KUKA KRL program: EPS_2_251580_SMH02_A_20251111081754.src

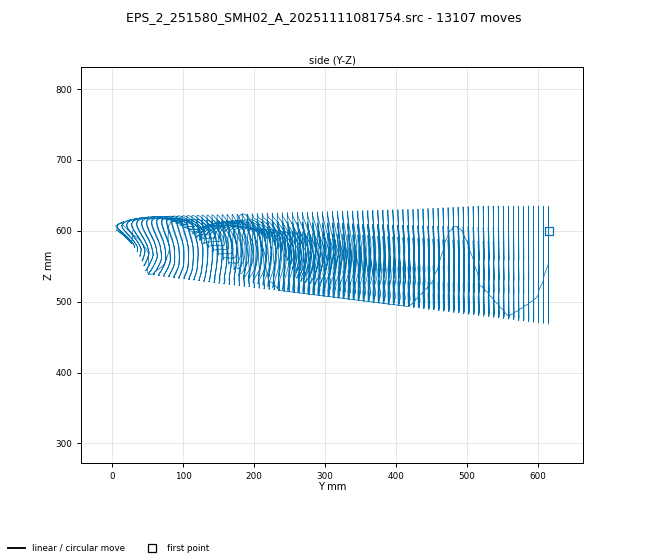
[picture p0: tool path of EPS_2_251580_SMH02_A_20251111081754.src, 13107 of 13109 moves have a stored position in this frame; points joined in program order, loops and branches not executed]
&ACCESS RVP
&REL 4
&COMMENT QRS 19112012
&PARAM EDITMASK = *
DEF PART()
EXT BAS (BAS_COMMAND :IN,REAL :IN )
INT I
BAS (#INITMOV,0 )

;KUKA QRS Post kuka4.cps  Date:22-06-2017 !

File_ID=2902

QRS_PRE_INIT()

;Init var - Until changes are made in qrs_pre_init
Outlet_Square_prg=0
Inlet_1_Square_prg=0
Inlet_2_Square_prg=0
Inlet_3_Square_prg=0
Inlet_4_Square_prg=0
Inlet_5_Square_prg=0

Outlet_1={X 0.000, Y 520.000, Z 560.000, B 0.000, E1 0.000 }
Inlet_1={X 0.000, Y 523.590, Z 510.000, B 0.000, E1 90.000 }
Inlet_2={X 0.000, Y 522.160, Z 530.000, B 0.000, E1 146.000 }
Outlet_1_type=150
Inlet_1_type=150
Inlet_2_type=150
;QRS#1=Sidecore dimensions
;QRS#2=150-6" PVC SDR 28
;QRS#3=150-6" PVC SDR 28
;QRS#4=150-6" PVC SDR 28
;QRS#5=
;QRS#6=
;QRS#7=
;QRS#8=
;QRS#9=10-06 PSX
;QRS#10=10-06 PSX
;QRS#11=10-06 PSX
;QRS#12=
;QRS#13=
;QRS#14=
;QRS#15=
;QRS#16=1220x127x914 3'
;QRS#17=EPS Height
;QRS#18=635
;QRS#19=*
;QRS#20= UPDATED VERSION 22-06-2017
;QRS#21=*
Outlet_Square=070
Inlet_1_Square=070
Inlet_2_Square=070
Inlet_3_Square=0
Inlet_4_Square=0
Inlet_5_Square=0
Mill_Square=1
Outlet_Square_Prg=203
Inlet_1_Square_prg=203
Inlet_2_Square_prg=203

QRS_INIT()

$ADVANCE=5

; T1
PTP {E1 173.473,E2 173.473}
PTP {X 0,Y 615.499,A -85,B 0,C 180,E1 173.473,E2 173.473,E3 0,E4 0,E5 0,E6 0}
QRS_SPEED_INIT()
LIN {X 0,Y 615.499,Z 600,A -85,B 0,C 180,E1 173.473,E2 173.473,E3 0,E4 0,E5 0,E6 0} C_VEL
LIN {X 0,Y 615.499,Z 569.968,A -85,B 0,C 180,E1 173.473,E2 173.473} C_VEL
LIN {X 0,Y 615.499,Z 557.271,A -85,B 0,C 180,E1 173.473,E2 173.473} C_VEL
LIN {X 0,Y 615.498,Z 555.824,A -85,B 0,C 180,E1 173.416,E2 173.416} C_VEL
LIN {X 0,Y 615.496,Z 547.552,A -85,B 0,C 180,E1 172.702,E2 172.702} C_VEL
LIN {X 0,Y 615.476,Z 537.678,A -85,B 0,C 180,E1 172.042,E2 172.042} C_VEL
LIN {X 0,Y 615.489,Z 529.919,A -85,B 0,C 180,E1 171.629,E2 171.629} C_VEL
LIN {X 0,Y 615.493,Z 521.057,A -85,B 0,C 180,E1 171.257,E2 171.257} C_VEL
LIN {X 0,Y 615.492,Z 511.835,A -85,B 0,C 180,E1 170.967,E2 170.967} C_VEL
LIN {X 0,Y 615.489,Z 506.039,A -85,B 0,C 180,E1 170.822,E2 170.822} C_VEL
LIN {X 0,Y 615.478,Z 501.144,A -85,B 0,C 180,E1 168.139,E2 168.139} C_VEL
LIN {X 0,Y 615.493,Z 496.29,A -85,B 0,C 180,E1 165.451,E2 165.451} C_VEL
LIN {X 0,Y 615.49,Z 491.434,A -85,B 0,C 180,E1 162.73,E2 162.73} C_VEL
LIN {X 0,Y 615.491,Z 486.577,A -85,B 0,C 180,E1 159.967,E2 159.967} C_VEL
LIN {X 0,Y 615.477,Z 481.72,A -85,B 0,C 180,E1 157.155,E2 157.155} C_VEL
LIN {X 0,Y 615.486,Z 477.105,A -85,B 0,C 180,E1 154.432,E2 154.432} C_VEL
LIN {X 0,Y 615.496,Z 474.066,A -85,B 0,C 180,E1 152.501,E2 152.501} C_VEL
LIN {X 0,Y 615.489,Z 480.62,A -85,B 0,C 180,E1 149.84,E2 149.84} C_VEL
LIN {X 0,Y 615.489,Z 486.401,A -85,B 0,C 180,E1 147.543,E2 147.543} C_VEL
LIN {X 0,Y 615.488,Z 493.466,A -85,B 0,C 180,E1 144.785,E2 144.785} C_VEL
LIN {X 0,Y 615.484,Z 500.912,A -85,B 0,C 180,E1 141.931,E2 141.931} C_VEL
LIN {X 0,Y 615.483,Z 507.646,A -85,B 0,C 180,E1 139.393,E2 139.393} C_VEL
LIN {X 0,Y 615.497,Z 514.698,A -85,B 0,C 180,E1 136.756,E2 136.756} C_VEL
LIN {X 0,Y 615.483,Z 522.177,A -85,B 0,C 180,E1 133.997,E2 133.997} C_VEL
LIN {X 0,Y 615.485,Z 524.739,A -85,B 0,C 180,E1 133.109,E2 133.109} C_VEL
LIN {X 0,Y 615.497,Z 537.239,A -85,B 0,C 180,E1 132.785,E2 132.785} C_VEL
LIN {X 0,Y 615.477,Z 546.369,A -85,B 0,C 180,E1 132.441,E2 132.441} C_VEL
LIN {X 0,Y 615.481,Z 555.26,A -85,B 0,C 180,E1 132.003,E2 132.003} C_VEL
LIN {X 0,Y 615.489,Z 562.693,A -85,B 0,C 180,E1 131.549,E2 131.549} C_VEL
LIN {X 0,Y 615.499,Z 570.437,A -85,B 0,C 180,E1 130.972,E2 130.972} C_VEL
LIN {X 0,Y 615.495,Z 577.327,A -85,B 0,C 180,E1 130.348,E2 130.348} C_VEL
LIN {X 0,Y 615.498,Z 584.294,A -85,B 0,C 180,E1 129.577,E2 129.577} C_VEL
LIN {X 0,Y 615.497,Z 590.588,A -85,B 0,C 180,E1 128.694,E2 128.694} C_VEL
LIN {X 0,Y 615.495,Z 594.491,A -85,B 0,C 180,E1 128.013,E2 128.013} C_VEL
LIN {X 0,Y 615.492,Z 598.012,A -85,B 0,C 180,E1 127.242,E2 127.242} C_VEL
LIN {X 0,Y 615.49,Z 600.84,A -85,B 0,C 180,E1 126.425,E2 126.425} C_VEL
LIN {X 0,Y 615.493,Z 602.8,A -85,B 0,C 180,E1 125.616,E2 125.616} C_VEL
LIN {X 0,Y 615.498,Z 604.058,A -85,B 0,C 180,E1 124.702,E2 124.702} C_VEL
LIN {X 0,Y 615.493,Z 604.378,A -85,B 0,C 180,E1 124.022,E2 124.022} C_VEL
LIN {X 0,Y 615.494,Z 604.074,A -85,B 0,C 180,E1 123.236,E2 123.236} C_VEL
LIN {X 0,Y 615.489,Z 602.87,A -85,B 0,C 180,E1 122.331,E2 122.331} C_VEL
LIN {X 0,Y 615.495,Z 601.344,A -85,B 0,C 180,E1 121.685,E2 121.685} C_VEL
LIN {X 0,Y 615.489,Z 597.454,A -85,B 0,C 180,E1 120.539,E2 120.539} C_VEL
LIN {X 0,Y 615.494,Z 592.819,A -85,B 0,C 180,E1 119.601,E2 119.601} C_VEL
LIN {X 0,Y 615.499,Z 588.063,A -85,B 0,C 180,E1 118.844,E2 118.844} C_VEL
LIN {X 0,Y 615.497,Z 583.01,A -85,B 0,C 180,E1 118.183,E2 118.183} C_VEL
LIN {X 0,Y 615.497,Z 577.153,A -85,B 0,C 180,E1 117.545,E2 117.545} C_VEL
LIN {X 0,Y 615.498,Z 569.916,A -85,B 0,C 180,E1 116.895,E2 116.895} C_VEL
LIN {X 0,Y 615.478,Z 562.594,A -85,B 0,C 180,E1 116.354,E2 116.354} C_VEL
LIN {X 0,Y 615.488,Z 553.468,A -85,B 0,C 180,E1 115.807,E2 115.807} C_VEL
LIN {X 0,Y 615.485,Z 541.734,A -85,B 0,C 180,E1 115.28,E2 115.28} C_VEL
LIN {X 0,Y 615.496,Z 532.824,A -85,B 0,C 180,E1 114.992,E2 114.992} C_VEL
LIN {X 0,Y 615.494,Z 524.808,A -85,B 0,C 180,E1 114.789,E2 114.789} C_VEL
LIN {X 0,Y 615.482,Z 518.038,A -85,B 0,C 180,E1 112.137,E2 112.137} C_VEL
LIN {X 0,Y 615.485,Z 510.962,A -85,B 0,C 180,E1 109.338,E2 109.338} C_VEL
LIN {X 0,Y 615.48,Z 504.089,A -85,B 0,C 180,E1 106.587,E2 106.587} C_VEL
LIN {X 0,Y 615.495,Z 497.407,A -85,B 0,C 180,E1 103.874,E2 103.874} C_VEL
LIN {X 0,Y 615.486,Z 490.182,A -85,B 0,C 180,E1 100.887,E2 100.887} C_VEL
LIN {X 0,Y 615.483,Z 484.608,A -85,B 0,C 180,E1 98.537,E2 98.537} C_VEL
LIN {X 0,Y 615.493,Z 478.479,A -85,B 0,C 180,E1 95.899,E2 95.899} C_VEL
LIN {X 0,Y 615.481,Z 472.517,A -85,B 0,C 180,E1 93.273,E2 93.273} C_VEL
LIN {X 0,Y 615.478,Z 468.511,A -85,B 0,C 180,E1 91.473,E2 91.473} C_VEL
LIN {X 0,Y 615.48,Z 468.51,A -85,B 0,C 180,E1 88.692,E2 88.692} C_VEL
LIN {X 0,Y 615.488,Z 468.512,A -85,B 0,C 180,E1 86.072,E2 86.072} C_VEL
LIN {X 0,Y 615.49,Z 468.512,A -85,B 0,C 180,E1 83.42,E2 83.42} C_VEL
LIN {X 0,Y 615.48,Z 468.511,A -85,B 0,C 180,E1 80.801,E2 80.801} C_VEL
LIN {X 0,Y 615.49,Z 468.508,A -85,B 0,C 180,E1 78.14,E2 78.14} C_VEL
LIN {X 0,Y 615.487,Z 468.512,A -85,B 0,C 180,E1 75.451,E2 75.451} C_VEL
LIN {X 0,Y 615.488,Z 468.511,A -85,B 0,C 180,E1 72.73,E2 72.73} C_VEL
LIN {X 0,Y 615.488,Z 468.508,A -85,B 0,C 180,E1 69.968,E2 69.968} C_VEL
LIN {X 0,Y 615.489,Z 468.512,A -85,B 0,C 180,E1 67.156,E2 67.156} C_VEL
LIN {X 0,Y 615.495,Z 468.507,A -85,B 0,C 180,E1 64.285,E2 64.285} C_VEL
LIN {X 0,Y 615.484,Z 468.511,A -85,B 0,C 180,E1 61.342,E2 61.342} C_VEL
LIN {X 0,Y 615.495,Z 468.51,A -85,B 0,C 180,E1 58.913,E2 58.913} C_VEL
LIN {X 0,Y 615.49,Z 468.513,A -85,B 0,C 180,E1 56.466,E2 56.466} C_VEL
LIN {X 0,Y 615.494,Z 468.511,A -85,B 0,C 180,E1 54.166,E2 54.166} C_VEL
LIN {X 0,Y 615.493,Z 468.509,A -85,B 0,C 180,E1 51.932,E2 51.932} C_VEL
LIN {X 0,Y 615.485,Z 468.514,A -85,B 0,C 180,E1 49.394,E2 49.394} C_VEL
LIN {X 0,Y 615.492,Z 468.511,A -85,B 0,C 180,E1 46.756,E2 46.756} C_VEL
LIN {X 0,Y 615.484,Z 468.509,A -85,B 0,C 180,E1 43.998,E2 43.998} C_VEL
LIN {X 0,Y 615.495,Z 468.512,A -85,B 0,C 180,E1 41.096,E2 41.096} C_VEL
LIN {X 0,Y 615.481,Z 468.512,A -85,B 0,C 180,E1 38.905,E2 38.905} C_VEL
LIN {X 0,Y 615.488,Z 468.512,A -85,B 0,C 180,E1 36.425,E2 36.425} C_VEL
LIN {X 0,Y 615.485,Z 468.509,A -85,B 0,C 180,E1 33.535,E2 33.535} C_VEL
LIN {X 0,Y 615.479,Z 468.51,A -85,B 0,C 180,E1 30.92,E2 30.92} C_VEL
LIN {X 0,Y 615.492,Z 468.507,A -85,B 0,C 180,E1 28.452,E2 28.452} C_VEL
LIN {X 0,Y 615.495,Z 468.512,A -85,B 0,C 180,E1 25.571,E2 25.571} C_VEL
LIN {X 0,Y 615.48,Z 468.51,A -85,B 0,C 180,E1 22.845,E2 22.845} C_VEL
LIN {X 0,Y 615.488,Z 468.51,A -85,B 0,C 180,E1 20.033,E2 20.033} C_VEL
LIN {X 0,Y 615.49,Z 468.512,A -85,B 0,C 180,E1 17.27,E2 17.27} C_VEL
LIN {X 0,Y 615.494,Z 468.507,A -85,B 0,C 180,E1 14.549,E2 14.549} C_VEL
LIN {X 0,Y 615.48,Z 468.511,A -85,B 0,C 180,E1 11.861,E2 11.861} C_VEL
LIN {X 0,Y 615.486,Z 468.514,A -85,B 0,C 180,E1 9.199,E2 9.199} C_VEL
LIN {X 0,Y 615.497,Z 468.509,A -85,B 0,C 180,E1 6.557,E2 6.557} C_VEL
LIN {X 0,Y 615.479,Z 468.51,A -85,B 0,C 180,E1 3.929,E2 3.929} C_VEL
LIN {X 0,Y 615.487,Z 468.508,A -85,B 0,C 180,E1 1.309,E2 1.309} C_VEL
LIN {X 0,Y 615.485,Z 468.512,A -85,B 0,C 180,E1 -1.309,E2 -1.309} C_VEL
LIN {X 0,Y 615.489,Z 468.514,A -85,B 0,C 180,E1 -3.928,E2 -3.928} C_VEL
LIN {X 0,Y 615.491,Z 468.508,A -85,B 0,C 180,E1 -6.584,E2 -6.584} C_VEL
LIN {X 0,Y 615.483,Z 468.509,A -85,B 0,C 180,E1 -9.199,E2 -9.199} C_VEL
LIN {X 0,Y 615.488,Z 468.51,A -85,B 0,C 180,E1 -11.861,E2 -11.861} C_VEL
LIN {X 0,Y 615.491,Z 468.514,A -85,B 0,C 180,E1 -14.549,E2 -14.549} C_VEL
LIN {X 0,Y 615.495,Z 468.507,A -85,B 0,C 180,E1 -17.27,E2 -17.27} C_VEL
LIN {X 0,Y 615.479,Z 468.511,A -85,B 0,C 180,E1 -20.033,E2 -20.033} C_VEL
LIN {X 0,Y 615.493,Z 468.512,A -85,B 0,C 180,E1 -22.844,E2 -22.844} C_VEL
LIN {X 0,Y 615.48,Z 468.51,A -85,B 0,C 180,E1 -25.716,E2 -25.716} C_VEL
LIN {X 0,Y 615.492,Z 468.514,A -85,B 0,C 180,E1 -28.658,E2 -28.658} C_VEL
LIN {X 0,Y 615.49,Z 468.514,A -85,B 0,C 180,E1 -31.087,E2 -31.087} C_VEL
LIN {X 0,Y 615.486,Z 468.513,A -85,B 0,C 180,E1 -33.535,E2 -33.535} C_VEL
LIN {X 0,Y 615.488,Z 468.508,A -85,B 0,C 180,E1 -36.425,E2 -36.425} C_VEL
LIN {X 0,Y 615.482,Z 468.512,A -85,B 0,C 180,E1 -39.062,E2 -39.062} C_VEL
LIN {X 0,Y 615.494,Z 468.51,A -85,B 0,C 180,E1 -41.473,E2 -41.473} C_VEL
LIN {X 0,Y 615.492,Z 468.512,A -85,B 0,C 180,E1 -44.149,E2 -44.149} C_VEL
LIN {X 0,Y 615.485,Z 468.509,A -85,B 0,C 180,E1 -46.953,E2 -46.953} C_VEL
LIN {X 0,Y 615.498,Z 468.512,A -85,B 0,C 180,E1 -49.91,E2 -49.91} C_VEL
LIN {X 0,Y 615.481,Z 468.51,A -85,B 0,C 180,E1 -52.758,E2 -52.758} C_VEL
LIN {X 0,Y 615.495,Z 468.506,A -85,B 0,C 180,E1 -55.298,E2 -55.298} C_VEL
LIN {X 0,Y 615.477,Z 468.51,A -85,B 0,C 180,E1 -57.671,E2 -57.671} C_VEL
LIN {X 0,Y 615.492,Z 468.707,A -85,B 0,C 180,E1 -59.081,E2 -59.081} C_VEL
LIN {X 0,Y 615.477,Z 477.608,A -85,B 0,C 180,E1 -61.552,E2 -61.552} C_VEL
LIN {X 0,Y 615.489,Z 487.691,A -85,B 0,C 180,E1 -64.285,E2 -64.285} C_VEL
LIN {X 0,Y 615.489,Z 498.525,A -85,B 0,C 180,E1 -67.156,E2 -67.156} C_VEL
LIN {X 0,Y 615.485,Z 509.354,A -85,B 0,C 180,E1 -69.968,E2 -69.968} C_VEL
LIN {X 0,Y 615.477,Z 520.179,A -85,B 0,C 180,E1 -72.73,E2 -72.73} C_VEL
LIN {X 0,Y 615.493,Z 530.988,A -85,B 0,C 180,E1 -75.451,E2 -75.451} C_VEL
LIN {X 0,Y 615.488,Z 541.8,A -85,B 0,C 180,E1 -78.14,E2 -78.14} C_VEL
LIN {X 0,Y 615.481,Z 552.598,A -85,B 0,C 180,E1 -80.801,E2 -80.801} C_VEL
LIN {X 0,Y 615.495,Z 566.17,A -85,B 0,C 180,E1 -81.133,E2 -81.133} C_VEL
LIN {X 0,Y 615.479,Z 575.233,A -85,B 0,C 180,E1 -81.464,E2 -81.464} C_VEL
LIN {X 0,Y 615.487,Z 583.917,A -85,B 0,C 180,E1 -81.877,E2 -81.877} C_VEL
LIN {X 0,Y 615.48,Z 592.206,A -85,B 0,C 180,E1 -82.372,E2 -82.372} C_VEL
LIN {X 0,Y 615.499,Z 599.937,A -85,B 0,C 180,E1 -82.942,E2 -82.942} C_VEL
LIN {X 0,Y 615.498,Z 605.649,A -85,B 0,C 180,E1 -83.444,E2 -83.444} C_VEL
LIN {X 0,Y 615.499,Z 611.924,A -85,B 0,C 180,E1 -84.102,E2 -84.102} C_VEL
LIN {X 0,Y 615.496,Z 617.138,A -85,B 0,C 180,E1 -84.759,E2 -84.759} C_VEL
LIN {X 0,Y 615.497,Z 621.484,A -85,B 0,C 180,E1 -85.416,E2 -85.416} C_VEL
LIN {X 0,Y 615.492,Z 626.605,A -85,B 0,C 180,E1 -86.4,E2 -86.4} C_VEL
LIN {X 0,Y 615.494,Z 629.221,A -85,B 0,C 180,E1 -87.055,E2 -87.055} C_VEL
LIN {X 0,Y 615.497,Z 632.086,A -85,B 0,C 180,E1 -88.037,E2 -88.037} C_VEL
LIN {X 0,Y 615.494,Z 633.33,A -85,B 0,C 180,E1 -88.692,E2 -88.692} C_VEL
LIN {X 0,Y 615.494,Z 634.104,A -85,B 0,C 180,E1 -89.346,E2 -89.346} C_VEL
LIN {X 0,Y 615.491,Z 634.389,A -85,B 0,C 180,E1 -90,E2 -90} C_VEL
LIN {X 0,Y 615.494,Z 634.104,A -85,B 0,C 180,E1 -90.655,E2 -90.655} C_VEL
LIN {X 0,Y 615.494,Z 633.329,A -85,B 0,C 180,E1 -91.309,E2 -91.309} C_VEL
LIN {X 0,Y 615.497,Z 632.085,A -85,B 0,C 180,E1 -91.963,E2 -91.963} C_VEL
LIN {X 0,Y 615.494,Z 629.218,A -85,B 0,C 180,E1 -92.946,E2 -92.946} C_VEL
LIN {X 0,Y 615.492,Z 626.602,A -85,B 0,C 180,E1 -93.601,E2 -93.601} C_VEL
LIN {X 0,Y 615.496,Z 621.48,A -85,B 0,C 180,E1 -94.585,E2 -94.585} C_VEL
LIN {X 0,Y 615.495,Z 615.966,A -85,B 0,C 180,E1 -95.406,E2 -95.406} C_VEL
LIN {X 0,Y 615.498,Z 609.015,A -85,B 0,C 180,E1 -96.228,E2 -96.228} C_VEL
LIN {X 0,Y 615.498,Z 601.856,A -85,B 0,C 180,E1 -96.901,E2 -96.901} C_VEL
LIN {X 0,Y 615.477,Z 594.619,A -85,B 0,C 180,E1 -97.463,E2 -97.463} C_VEL
LIN {X 0,Y 615.492,Z 586.863,A -85,B 0,C 180,E1 -97.958,E2 -97.958} C_VEL
LIN {X 0,Y 615.478,Z 578.911,A -85,B 0,C 180,E1 -98.372,E2 -98.372} C_VEL
LIN {X 0,Y 615.485,Z 569.748,A -85,B 0,C 180,E1 -98.744,E2 -98.744} C_VEL
LIN {X 0,Y 615.493,Z 561.68,A -85,B 0,C 180,E1 -98.992,E2 -98.992} C_VEL
LIN {X 0,Y 615.48,Z 552.911,A -85,B 0,C 180,E1 -99.199,E2 -99.199} C_VEL
LIN {X 0,Y 615.488,Z 542.765,A -85,B 0,C 180,E1 -101.861,E2 -101.861} C_VEL
LIN {X 0,Y 615.485,Z 532.6,A -85,B 0,C 180,E1 -104.549,E2 -104.549} C_VEL
LIN {X 0,Y 615.477,Z 522.449,A -85,B 0,C 180,E1 -107.271,E2 -107.271} C_VEL
LIN {X 0,Y 615.486,Z 512.267,A -85,B 0,C 180,E1 -110.033,E2 -110.033} C_VEL
LIN {X 0,Y 615.488,Z 502.099,A -85,B 0,C 180,E1 -112.845,E2 -112.845} C_VEL
LIN {X 0,Y 615.489,Z 491.908,A -85,B 0,C 180,E1 -115.716,E2 -115.716} C_VEL
LIN {X 0,Y 615.477,Z 482.445,A -85,B 0,C 180,E1 -118.449,E2 -118.449} C_VEL
LIN {X 0,Y 615.488,Z 473.518,A -85,B 0,C 180,E1 -121.086,E2 -121.086} C_VEL
LIN {X 0,Y 615.493,Z 468.504,A -85,B 0,C 180,E1 -122.652,E2 -122.652} C_VEL
LIN {X 0,Y 615.499,Z 468.5,A -85,B 0,C 180,E1 -124.815,E2 -124.815} C_VEL
LIN {X 0,Y 615.483,Z 468.511,A -85,B 0,C 180,E1 -127.243,E2 -127.243} C_VEL
LIN {X 0,Y 615.486,Z 468.511,A -85,B 0,C 180,E1 -130.089,E2 -130.089} C_VEL
LIN {X 0,Y 615.49,Z 468.505,A -85,B 0,C 180,E1 -133.048,E2 -133.048} C_VEL
LIN {X 0,Y 615.484,Z 468.504,A -85,B 0,C 180,E1 -136.003,E2 -136.003} C_VEL
LIN {X 0,Y 615.494,Z 468.505,A -85,B 0,C 180,E1 -138.527,E2 -138.527} C_VEL
LIN {X 0,Y 615.49,Z 468.507,A -85,B 0,C 180,E1 -141.096,E2 -141.096} C_VEL
LIN {X 0,Y 615.488,Z 468.503,A -85,B 0,C 180,E1 -143.575,E2 -143.575} C_VEL
LIN {X 0,Y 615.494,Z 468.506,A -85,B 0,C 180,E1 -146.465,E2 -146.465} C_VEL
LIN {X 0,Y 615.493,Z 468.607,A -85,B 0,C 180,E1 -147.669,E2 -147.669} C_VEL
LIN {X 0,Y 615.477,Z 472.359,A -85,B 0,C 180,E1 -150.208,E2 -150.208} C_VEL
LIN {X 0,Y 615.483,Z 476.576,A -85,B 0,C 180,E1 -152.956,E2 -152.956} C_VEL
LIN {X 0,Y 615.489,Z 480.934,A -85,B 0,C 180,E1 -155.728,E2 -155.728} C_VEL
LIN {X 0,Y 615.498,Z 485.495,A -85,B 0,C 180,E1 -158.569,E2 -158.569} C_VEL
LIN {X 0,Y 615.485,Z 490.138,A -85,B 0,C 180,E1 -161.397,E2 -161.397} C_VEL
LIN {X 0,Y 615.486,Z 494.622,A -85,B 0,C 180,E1 -164.095,E2 -164.095} C_VEL
LIN {X 0,Y 615.487,Z 499.189,A -85,B 0,C 180,E1 -166.799,E2 -166.799} C_VEL
LIN {X 0,Y 615.497,Z 503.742,A -85,B 0,C 180,E1 -169.473,E2 -169.473} C_VEL
LIN {X 0,Y 615.492,Z 506.209,A -85,B 0,C 180,E1 -170.905,E2 -170.905} C_VEL
LIN {X 0,Y 615.489,Z 518.455,A -85,B 0,C 180,E1 -171.257,E2 -171.257} C_VEL
LIN {X 0,Y 615.485,Z 526.066,A -85,B 0,C 180,E1 -171.546,E2 -171.546} C_VEL
LIN {X 0,Y 615.477,Z 534.588,A -85,B 0,C 180,E1 -171.959,E2 -171.959} C_VEL
LIN {X 0,Y 615.491,Z 542.749,A -85,B 0,C 180,E1 -172.455,E2 -172.455} C_VEL
LIN {X 0,Y 615.498,Z 549.392,A -85,B 0,C 180,E1 -172.942,E2 -172.942} C_VEL
LIN {X 0,Y 615.498,Z 555.185,A -85,B 0,C 180,E1 -173.443,E2 -173.443} C_VEL
LIN {X 0,Y 615.499,Z 561.535,A -85,B 0,C 180,E1 -174.102,E2 -174.102} C_VEL
LIN {X 0,Y 615.495,Z 567.984,A -85,B 0,C 180,E1 -174.923,E2 -174.923} C_VEL
LIN {X 0,Y 615.492,Z 573.123,A -85,B 0,C 180,E1 -175.744,E2 -175.744} C_VEL
LIN {X 0,Y 615.495,Z 577.886,A -85,B 0,C 180,E1 -176.727,E2 -176.727} C_VEL
LIN {X 0,Y 615.493,Z 580.2,A -85,B 0,C 180,E1 -177.382,E2 -177.382} C_VEL
LIN {X 0,Y 615.494,Z 581.977,A -85,B 0,C 180,E1 -178.037,E2 -178.037} C_VEL
LIN {X 0,Y 615.496,Z 583.265,A -85,B 0,C 180,E1 -178.691,E2 -178.691} C_VEL
LIN {X 0,Y 615.492,Z 584.083,A -85,B 0,C 180,E1 -179.346,E2 -179.346} C_VEL
LIN {X 0,Y 615.49,Z 584.385,A -85,B 0,C 180,E1 -180,E2 -180} C_VEL
LIN {X 0,Y 615.494,Z 584.124,A -85,B 0,C 180,E1 -180.654,E2 -180.654} C_VEL
LIN {X 0,Y 615.494,Z 583.393,A -85,B 0,C 180,E1 -181.309,E2 -181.309} C_VEL
LIN {X 0,Y 615.498,Z 582.194,A -85,B 0,C 180,E1 -181.963,E2 -181.963} C_VEL
LIN {X 0,Y 615.49,Z 579.376,A -85,B 0,C 180,E1 -182.945,E2 -182.945} C_VEL
LIN {X 0,Y 615.496,Z 576.809,A -85,B 0,C 180,E1 -183.601,E2 -183.601} C_VEL
LIN {X 0,Y 615.498,Z 571.742,A -85,B 0,C 180,E1 -184.585,E2 -184.585} C_VEL
LIN {X 0,Y 615.496,Z 566.287,A -85,B 0,C 180,E1 -185.405,E2 -185.405} C_VEL
LIN {X 0,Y 615.497,Z 559.452,A -85,B 0,C 180,E1 -186.227,E2 -186.227} C_VEL
LIN {X 0,Y 615.498,Z 555.824,A -85,B 0,C 180,E1 -186.584,E2 -186.584} C_VEL
LIN {X 0,Y 614.837,Z 551.743,A -85,B 0,C 180,E1 -186.977,E2 -186.977} C_VEL
LIN {X 0,Y 611.991,Z 544.71,A -85,B 0,C 180,E1 -187.582,E2 -187.582} C_VEL
LIN {X 0,Y 609.148,Z 537.088,A -85,B 0,C 180,E1 -188.113,E2 -188.113} C_VEL
LIN {X 0,Y 608.482,Z 531.993,A -85,B 0,C 180,E1 -188.386,E2 -188.386} C_VEL
LIN {X 0,Y 608.484,Z 521.382,A -85,B 0,C 180,E1 -188.845,E2 -188.845} C_VEL
LIN {X 0,Y 608.509,Z 511.365,A -85,B 0,C 180,E1 -189.159,E2 -189.159} C_VEL
LIN {X 0,Y 608.424,Z 506.525,A -85,B 0,C 180,E1 -189.286,E2 -189.286} C_VEL
LIN {X 0,Y 608.42,Z 501.596,A -85,B 0,C 180,E1 -192.001,E2 -192.001} C_VEL
LIN {X 0,Y 608.421,Z 496.706,A -85,B 0,C 180,E1 -194.722,E2 -194.722} C_VEL
LIN {X 0,Y 608.434,Z 491.815,A -85,B 0,C 180,E1 -197.477,E2 -197.477} C_VEL
LIN {X 0,Y 608.431,Z 486.924,A -85,B 0,C 180,E1 -200.275,E2 -200.275} C_VEL
LIN {X 0,Y 608.43,Z 482.033,A -85,B 0,C 180,E1 -203.125,E2 -203.125} C_VEL
LIN {X 0,Y 608.451,Z 477.141,A -85,B 0,C 180,E1 -206.035,E2 -206.035} C_VEL
LIN {X 0,Y 608.46,Z 474.892,A -85,B 0,C 180,E1 -207.421,E2 -207.421} C_VEL
LIN {X 0,Y 608.45,Z 481.115,A -85,B 0,C 180,E1 -209.968,E2 -209.968} C_VEL
LIN {X 0,Y 608.464,Z 487.492,A -85,B 0,C 180,E1 -212.522,E2 -212.522} C_VEL
LIN {X 0,Y 608.454,Z 494.511,A -85,B 0,C 180,E1 -215.277,E2 -215.277} C_VEL
LIN {X 0,Y 608.426,Z 500.923,A -85,B 0,C 180,E1 -217.749,E2 -217.749} C_VEL
LIN {X 0,Y 608.435,Z 507.701,A -85,B 0,C 180,E1 -220.327,E2 -220.327} C_VEL
LIN {X 0,Y 608.451,Z 514.716,A -85,B 0,C 180,E1 -222.96,E2 -222.96} C_VEL
LIN {X 0,Y 608.433,Z 522.201,A -85,B 0,C 180,E1 -225.738,E2 -225.738} C_VEL
LIN {X 0,Y 608.434,Z 525.065,A -85,B 0,C 180,E1 -226.781,E2 -226.781} C_VEL
LIN {X 0,Y 608.489,Z 536.811,A -85,B 0,C 180,E1 -227.086,E2 -227.086} C_VEL
LIN {X 0,Y 608.472,Z 546.89,A -85,B 0,C 180,E1 -227.47,E2 -227.47} C_VEL
LIN {X 0,Y 608.458,Z 554.986,A -85,B 0,C 180,E1 -227.869,E2 -227.869} C_VEL
LIN {X 0,Y 608.48,Z 562.562,A -85,B 0,C 180,E1 -228.33,E2 -228.33} C_VEL
LIN {X 0,Y 608.484,Z 570.681,A -85,B 0,C 180,E1 -228.935,E2 -228.935} C_VEL
LIN {X 0,Y 608.455,Z 578.951,A -85,B 0,C 180,E1 -229.697,E2 -229.697} C_VEL
LIN {X 0,Y 608.456,Z 586.305,A -85,B 0,C 180,E1 -230.559,E2 -230.559} C_VEL
LIN {X 0,Y 608.432,Z 591.996,A -85,B 0,C 180,E1 -231.409,E2 -231.409} C_VEL
LIN {X 0,Y 608.437,Z 596.455,A -85,B 0,C 180,E1 -232.251,E2 -232.251} C_VEL
LIN {X 0,Y 608.432,Z 599.848,A -85,B 0,C 180,E1 -233.083,E2 -233.083} C_VEL
LIN {X 0,Y 608.423,Z 602.434,A -85,B 0,C 180,E1 -233.958,E2 -233.958} C_VEL
LIN {X 0,Y 608.422,Z 604.469,A -85,B 0,C 180,E1 -235.098,E2 -235.098} C_VEL
LIN {X 0,Y 608.418,Z 604.892,A -85,B 0,C 180,E1 -236.326,E2 -236.326} C_VEL
LIN {X 0,Y 608.416,Z 603.77,A -85,B 0,C 180,E1 -237.485,E2 -237.485} C_VEL
LIN {X 0,Y 608.449,Z 600.97,A -85,B 0,C 180,E1 -238.682,E2 -238.682} C_VEL
LIN {X 0,Y 608.437,Z 598.217,A -85,B 0,C 180,E1 -239.453,E2 -239.453} C_VEL
LIN {X 0,Y 608.459,Z 593.559,A -85,B 0,C 180,E1 -240.41,E2 -240.41} C_VEL
LIN {X 0,Y 608.462,Z 588.551,A -85,B 0,C 180,E1 -241.214,E2 -241.214} C_VEL
LIN {X 0,Y 608.453,Z 583.142,A -85,B 0,C 180,E1 -241.921,E2 -241.921} C_VEL
LIN {X 0,Y 608.47,Z 578.039,A -85,B 0,C 180,E1 -242.483,E2 -242.483} C_VEL
LIN {X 0,Y 608.464,Z 571.669,A -85,B 0,C 180,E1 -243.074,E2 -243.074} C_VEL
LIN {X 0,Y 608.46,Z 563.615,A -85,B 0,C 180,E1 -243.688,E2 -243.688} C_VEL
LIN {X 0,Y 608.463,Z 556.073,A -85,B 0,C 180,E1 -244.16,E2 -244.16} C_VEL
LIN {X 0,Y 608.484,Z 548.335,A -85,B 0,C 180,E1 -244.554,E2 -244.554} C_VEL
LIN {X 0,Y 608.485,Z 540.291,A -85,B 0,C 180,E1 -244.883,E2 -244.883} C_VEL
LIN {X 0,Y 608.509,Z 531.4,A -85,B 0,C 180,E1 -245.158,E2 -245.158} C_VEL
LIN {X 0,Y 608.432,Z 525.267,A -85,B 0,C 180,E1 -245.314,E2 -245.314} C_VEL
LIN {X 0,Y 608.435,Z 519.472,A -85,B 0,C 180,E1 -247.593,E2 -247.593} C_VEL
LIN {X 0,Y 608.431,Z 512.328,A -85,B 0,C 180,E1 -250.428,E2 -250.428} C_VEL
LIN {X 0,Y 608.442,Z 505.393,A -85,B 0,C 180,E1 -253.215,E2 -253.215} C_VEL
LIN {X 0,Y 608.443,Z 498.583,A -85,B 0,C 180,E1 -255.993,E2 -255.993} C_VEL
LIN {X 0,Y 608.446,Z 492.122,A -85,B 0,C 180,E1 -258.675,E2 -258.675} C_VEL
LIN {X 0,Y 608.454,Z 485.77,A -85,B 0,C 180,E1 -261.364,E2 -261.364} C_VEL
LIN {X 0,Y 608.467,Z 479.6,A -85,B 0,C 180,E1 -264.033,E2 -264.033} C_VEL
LIN {X 0,Y 608.448,Z 473.615,A -85,B 0,C 180,E1 -266.689,E2 -266.689} C_VEL
LIN {X 0,Y 608.444,Z 469.509,A -85,B 0,C 180,E1 -268.428,E2 -268.428} C_VEL
LIN {X 0,Y 608.482,Z 469.506,A -85,B 0,C 180,E1 -270.661,E2 -270.661} C_VEL
LIN {X 0,Y 608.475,Z 469.504,A -85,B 0,C 180,E1 -273.31,E2 -273.31} C_VEL
LIN {X 0,Y 608.468,Z 469.505,A -85,B 0,C 180,E1 -275.966,E2 -275.966} C_VEL
LIN {X 0,Y 608.455,Z 469.509,A -85,B 0,C 180,E1 -278.636,E2 -278.636} C_VEL
LIN {X 0,Y 608.485,Z 469.505,A -85,B 0,C 180,E1 -281.323,E2 -281.323} C_VEL
LIN {X 0,Y 608.472,Z 469.505,A -85,B 0,C 180,E1 -284.037,E2 -284.037} C_VEL
LIN {X 0,Y 608.457,Z 469.507,A -85,B 0,C 180,E1 -286.784,E2 -286.784} C_VEL
LIN {X 0,Y 608.453,Z 469.509,A -85,B 0,C 180,E1 -289.57,E2 -289.57} C_VEL
LIN {X 0,Y 608.459,Z 469.506,A -85,B 0,C 180,E1 -292.406,E2 -292.406} C_VEL
LIN {X 0,Y 608.455,Z 469.507,A -85,B 0,C 180,E1 -294.571,E2 -294.571} C_VEL
LIN {X 0,Y 608.477,Z 469.504,A -85,B 0,C 180,E1 -297.207,E2 -297.207} C_VEL
LIN {X 0,Y 608.476,Z 469.507,A -85,B 0,C 180,E1 -299.973,E2 -299.973} C_VEL
LIN {X 0,Y 608.468,Z 469.508,A -85,B 0,C 180,E1 -302.523,E2 -302.523} C_VEL
LIN {X 0,Y 608.447,Z 469.508,A -85,B 0,C 180,E1 -305.277,E2 -305.277} C_VEL
LIN {X 0,Y 608.477,Z 469.504,A -85,B 0,C 180,E1 -307.745,E2 -307.745} C_VEL
LIN {X 0,Y 608.447,Z 469.508,A -85,B 0,C 180,E1 -310.328,E2 -310.328} C_VEL
LIN {X 0,Y 608.479,Z 469.505,A -85,B 0,C 180,E1 -313.31,E2 -313.31} C_VEL
LIN {X 0,Y 608.471,Z 469.505,A -85,B 0,C 180,E1 -316.131,E2 -316.131} C_VEL
LIN {X 0,Y 608.462,Z 469.508,A -85,B 0,C 180,E1 -318.824,E2 -318.824} C_VEL
LIN {X 0,Y 608.467,Z 469.508,A -85,B 0,C 180,E1 -321.412,E2 -321.412} C_VEL
LIN {X 0,Y 608.444,Z 469.509,A -85,B 0,C 180,E1 -323.954,E2 -323.954} C_VEL
LIN {X 0,Y 608.465,Z 469.507,A -85,B 0,C 180,E1 -326.329,E2 -326.329} C_VEL
LIN {X 0,Y 608.476,Z 469.505,A -85,B 0,C 180,E1 -328.727,E2 -328.727} C_VEL
LIN {X 0,Y 608.474,Z 469.504,A -85,B 0,C 180,E1 -331.379,E2 -331.379} C_VEL
LIN {X 0,Y 608.479,Z 469.507,A -85,B 0,C 180,E1 -334.277,E2 -334.277} C_VEL
LIN {X 0,Y 608.447,Z 469.51,A -85,B 0,C 180,E1 -336.876,E2 -336.876} C_VEL
LIN {X 0,Y 608.471,Z 469.506,A -85,B 0,C 180,E1 -339.319,E2 -339.319} C_VEL
LIN {X 0,Y 608.446,Z 469.508,A -85,B 0,C 180,E1 -341.828,E2 -341.828} C_VEL
LIN {X 0,Y 608.475,Z 469.505,A -85,B 0,C 180,E1 -344.594,E2 -344.594} C_VEL
LIN {X 0,Y 608.48,Z 469.507,A -85,B 0,C 180,E1 -347.323,E2 -347.323} C_VEL
LIN {X 0,Y 608.453,Z 469.508,A -85,B 0,C 180,E1 -350.023,E2 -350.023} C_VEL
LIN {X 0,Y 608.462,Z 469.506,A -85,B 0,C 180,E1 -352.701,E2 -352.701} C_VEL
LIN {X 0,Y 608.455,Z 469.508,A -85,B 0,C 180,E1 -355.362,E2 -355.362} C_VEL
LIN {X 0,Y 608.462,Z 469.509,A -85,B 0,C 180,E1 -358.014,E2 -358.014} C_VEL
LIN {X 0,Y 608.479,Z 469.504,A -85,B 0,C 180,E1 -360.662,E2 -360.662} C_VEL
LIN {X 0,Y 608.482,Z 469.503,A -85,B 0,C 180,E1 -363.311,E2 -363.311} C_VEL
LIN {X 0,Y 608.461,Z 469.507,A -85,B 0,C 180,E1 -365.967,E2 -365.967} C_VEL
LIN {X 0,Y 608.462,Z 469.509,A -85,B 0,C 180,E1 -368.636,E2 -368.636} C_VEL
LIN {X 0,Y 608.481,Z 469.504,A -85,B 0,C 180,E1 -371.324,E2 -371.324} C_VEL
LIN {X 0,Y 608.466,Z 469.505,A -85,B 0,C 180,E1 -374.037,E2 -374.037} C_VEL
LIN {X 0,Y 608.476,Z 469.507,A -85,B 0,C 180,E1 -376.783,E2 -376.783} C_VEL
LIN {X 0,Y 608.453,Z 469.508,A -85,B 0,C 180,E1 -379.571,E2 -379.571} C_VEL
LIN {X 0,Y 608.458,Z 469.507,A -85,B 0,C 180,E1 -382.477,E2 -382.477} C_VEL
LIN {X 0,Y 608.456,Z 469.507,A -85,B 0,C 180,E1 -384.571,E2 -384.571} C_VEL
LIN {X 0,Y 608.475,Z 469.505,A -85,B 0,C 180,E1 -387.207,E2 -387.207} C_VEL
LIN {X 0,Y 608.474,Z 469.507,A -85,B 0,C 180,E1 -389.973,E2 -389.973} C_VEL
LIN {X 0,Y 608.463,Z 469.507,A -85,B 0,C 180,E1 -392.523,E2 -392.523} C_VEL
LIN {X 0,Y 608.449,Z 469.507,A -85,B 0,C 180,E1 -395.277,E2 -395.277} C_VEL
LIN {X 0,Y 608.473,Z 469.505,A -85,B 0,C 180,E1 -397.746,E2 -397.746} C_VEL
LIN {X 0,Y 608.453,Z 469.509,A -85,B 0,C 180,E1 -400.33,E2 -400.33} C_VEL
LIN {X 0,Y 608.484,Z 469.503,A -85,B 0,C 180,E1 -403.311,E2 -403.311} C_VEL
LIN {X 0,Y 608.468,Z 469.506,A -85,B 0,C 180,E1 -406.131,E2 -406.131} C_VEL
LIN {X 0,Y 608.459,Z 469.509,A -85,B 0,C 180,E1 -408.824,E2 -408.824} C_VEL
LIN {X 0,Y 608.47,Z 469.506,A -85,B 0,C 180,E1 -411.413,E2 -411.413} C_VEL
LIN {X 0,Y 608.477,Z 469.504,A -85,B 0,C 180,E1 -413.951,E2 -413.951} C_VEL
LIN {X 0,Y 608.462,Z 469.506,A -85,B 0,C 180,E1 -416.33,E2 -416.33} C_VEL
LIN {X 0,Y 608.462,Z 469.531,A -85,B 0,C 180,E1 -418.912,E2 -418.912} C_VEL
LIN {X 0,Y 608.495,Z 478.299,A -85,B 0,C 180,E1 -421.376,E2 -421.376} C_VEL
LIN {X 0,Y 608.512,Z 488.872,A -85,B 0,C 180,E1 -424.271,E2 -424.271} C_VEL
LIN {X 0,Y 608.465,Z 499.983,A -85,B 0,C 180,E1 -427.237,E2 -427.237} C_VEL
LIN {X 0,Y 608.461,Z 509.494,A -85,B 0,C 180,E1 -429.726,E2 -429.726} C_VEL
LIN {X 0,Y 608.452,Z 520.365,A -85,B 0,C 180,E1 -432.524,E2 -432.524} C_VEL
LIN {X 0,Y 608.452,Z 531.236,A -85,B 0,C 180,E1 -435.279,E2 -435.279} C_VEL
LIN {X 0,Y 608.431,Z 542.107,A -85,B 0,C 180,E1 -438,E2 -438} C_VEL
LIN {X 0,Y 608.42,Z 552.978,A -85,B 0,C 180,E1 -440.694,E2 -440.694} C_VEL
LIN {X 0,Y 608.499,Z 566.491,A -85,B 0,C 180,E1 -441.03,E2 -441.03} C_VEL
LIN {X 0,Y 608.477,Z 575.541,A -85,B 0,C 180,E1 -441.365,E2 -441.365} C_VEL
LIN {X 0,Y 608.466,Z 584.238,A -85,B 0,C 180,E1 -441.783,E2 -441.783} C_VEL
LIN {X 0,Y 608.46,Z 592.547,A -85,B 0,C 180,E1 -442.284,E2 -442.284} C_VEL
LIN {X 0,Y 608.463,Z 600.405,A -85,B 0,C 180,E1 -442.868,E2 -442.868} C_VEL
LIN {X 0,Y 608.466,Z 607.359,A -85,B 0,C 180,E1 -443.496,E2 -443.496} C_VEL
LIN {X 0,Y 608.469,Z 615.194,A -85,B 0,C 180,E1 -444.366,E2 -444.366} C_VEL
LIN {X 0,Y 608.449,Z 621.029,A -85,B 0,C 180,E1 -445.197,E2 -445.197} C_VEL
LIN {X 0,Y 608.431,Z 625.632,A -85,B 0,C 180,E1 -446.026,E2 -446.026} C_VEL
LIN {X 0,Y 608.425,Z 628.623,A -85,B 0,C 180,E1 -446.689,E2 -446.689} C_VEL
LIN {X 0,Y 608.426,Z 630.932,A -85,B 0,C 180,E1 -447.352,E2 -447.352} C_VEL
LIN {X 0,Y 608.442,Z 632.679,A -85,B 0,C 180,E1 -448.015,E2 -448.015} C_VEL
LIN {X 0,Y 608.446,Z 633.934,A -85,B 0,C 180,E1 -448.677,E2 -448.677} C_VEL
LIN {X 0,Y 608.436,Z 634.714,A -85,B 0,C 180,E1 -449.339,E2 -449.339} C_VEL
LIN {X 0,Y 608.431,Z 635,A -85,B 0,C 180,E1 -450,E2 -450} C_VEL
LIN {X 0,Y 608.436,Z 634.713,A -85,B 0,C 180,E1 -450.662,E2 -450.662} C_VEL
LIN {X 0,Y 608.446,Z 633.933,A -85,B 0,C 180,E1 -451.324,E2 -451.324} C_VEL
LIN {X 0,Y 608.442,Z 632.677,A -85,B 0,C 180,E1 -451.986,E2 -451.986} C_VEL
LIN {X 0,Y 608.449,Z 629.785,A -85,B 0,C 180,E1 -452.98,E2 -452.98} C_VEL
LIN {X 0,Y 608.446,Z 627.144,A -85,B 0,C 180,E1 -453.643,E2 -453.643} C_VEL
LIN {X 0,Y 608.447,Z 621.983,A -85,B 0,C 180,E1 -454.638,E2 -454.638} C_VEL
LIN {X 0,Y 608.46,Z 616.427,A -85,B 0,C 180,E1 -455.468,E2 -455.468} C_VEL
LIN {X 0,Y 608.455,Z 608.67,A -85,B 0,C 180,E1 -456.376,E2 -456.376} C_VEL
LIN {X 0,Y 608.484,Z 601.411,A -85,B 0,C 180,E1 -457.049,E2 -457.049} C_VEL
LIN {X 0,Y 608.46,Z 593.755,A -85,B 0,C 180,E1 -457.634,E2 -457.634} C_VEL
LIN {X 0,Y 608.487,Z 585.713,A -85,B 0,C 180,E1 -458.134,E2 -458.134} C_VEL
LIN {X 0,Y 608.484,Z 577.381,A -85,B 0,C 180,E1 -458.552,E2 -458.552} C_VEL
LIN {X 0,Y 608.486,Z 568.878,A -85,B 0,C 180,E1 -458.887,E2 -458.887} C_VEL
LIN {X 0,Y 608.502,Z 559.571,A -85,B 0,C 180,E1 -459.159,E2 -459.159} C_VEL
LIN {X 0,Y 608.418,Z 553.301,A -85,B 0,C 180,E1 -459.307,E2 -459.307} C_VEL
LIN {X 0,Y 608.43,Z 543.082,A -85,B 0,C 180,E1 -462.001,E2 -462.001} C_VEL
LIN {X 0,Y 608.45,Z 532.864,A -85,B 0,C 180,E1 -464.721,E2 -464.721} C_VEL
LIN {X 0,Y 608.452,Z 522.645,A -85,B 0,C 180,E1 -467.477,E2 -467.477} C_VEL
LIN {X 0,Y 608.465,Z 512.426,A -85,B 0,C 180,E1 -470.274,E2 -470.274} C_VEL
LIN {X 0,Y 608.461,Z 503.486,A -85,B 0,C 180,E1 -472.764,E2 -472.764} C_VEL
LIN {X 0,Y 608.465,Z 494.543,A -85,B 0,C 180,E1 -475.301,E2 -475.301} C_VEL
LIN {X 0,Y 608.5,Z 485.602,A -85,B 0,C 180,E1 -477.89,E2 -477.89} C_VEL
LIN {X 0,Y 608.502,Z 476.661,A -85,B 0,C 180,E1 -480.543,E2 -480.543} C_VEL
LIN {X 0,Y 608.468,Z 469.505,A -85,B 0,C 180,E1 -482.774,E2 -482.774} C_VEL
LIN {X 0,Y 608.45,Z 469.509,A -85,B 0,C 180,E1 -485.278,E2 -485.278} C_VEL
LIN {X 0,Y 608.468,Z 469.502,A -85,B 0,C 180,E1 -487.747,E2 -487.747} C_VEL
LIN {X 0,Y 608.453,Z 469.509,A -85,B 0,C 180,E1 -490.329,E2 -490.329} C_VEL
LIN {X 0,Y 608.479,Z 469.506,A -85,B 0,C 180,E1 -493.31,E2 -493.31} C_VEL
LIN {X 0,Y 608.471,Z 469.503,A -85,B 0,C 180,E1 -496.131,E2 -496.131} C_VEL
LIN {X 0,Y 608.454,Z 469.504,A -85,B 0,C 180,E1 -498.823,E2 -498.823} C_VEL
LIN {X 0,Y 608.467,Z 469.504,A -85,B 0,C 180,E1 -501.76,E2 -501.76} C_VEL
LIN {X 0,Y 608.447,Z 469.505,A -85,B 0,C 180,E1 -503.955,E2 -503.955} C_VEL
LIN {X 0,Y 608.467,Z 469.507,A -85,B 0,C 180,E1 -506.33,E2 -506.33} C_VEL
LIN {X 0,Y 608.461,Z 469.506,A -85,B 0,C 180,E1 -507.478,E2 -507.478} C_VEL
LIN {X 0,Y 608.454,Z 471.029,A -85,B 0,C 180,E1 -508.732,E2 -508.732} C_VEL
LIN {X 0,Y 608.432,Z 474.98,A -85,B 0,C 180,E1 -511.388,E2 -511.388} C_VEL
LIN {X 0,Y 608.423,Z 479.46,A -85,B 0,C 180,E1 -514.289,E2 -514.289} C_VEL
LIN {X 0,Y 608.411,Z 483.546,A -85,B 0,C 180,E1 -516.874,E2 -516.874} C_VEL
LIN {X 0,Y 608.43,Z 488.141,A -85,B 0,C 180,E1 -519.725,E2 -519.725} C_VEL
LIN {X 0,Y 608.438,Z 492.736,A -85,B 0,C 180,E1 -522.523,E2 -522.523} C_VEL
LIN {X 0,Y 608.418,Z 497.331,A -85,B 0,C 180,E1 -525.278,E2 -525.278} C_VEL
LIN {X 0,Y 608.418,Z 501.927,A -85,B 0,C 180,E1 -527.999,E2 -527.999} C_VEL
LIN {X 0,Y 608.422,Z 506.702,A -85,B 0,C 180,E1 -530.798,E2 -530.798} C_VEL
LIN {X 0,Y 608.481,Z 518.799,A -85,B 0,C 180,E1 -531.155,E2 -531.155} C_VEL
LIN {X 0,Y 608.49,Z 526.392,A -85,B 0,C 180,E1 -531.448,E2 -531.448} C_VEL
LIN {X 0,Y 608.464,Z 534.919,A -85,B 0,C 180,E1 -531.866,E2 -531.866} C_VEL
LIN {X 0,Y 608.465,Z 543.104,A -85,B 0,C 180,E1 -532.367,E2 -532.367} C_VEL
LIN {X 0,Y 608.456,Z 550.868,A -85,B 0,C 180,E1 -532.951,E2 -532.951} C_VEL
LIN {X 0,Y 608.456,Z 558.235,A -85,B 0,C 180,E1 -533.627,E2 -533.627} C_VEL
LIN {X 0,Y 608.46,Z 566.111,A -85,B 0,C 180,E1 -534.532,E2 -534.532} C_VEL
LIN {X 0,Y 608.445,Z 571.725,A -85,B 0,C 180,E1 -535.362,E2 -535.362} C_VEL
LIN {X 0,Y 608.446,Z 576.941,A -85,B 0,C 180,E1 -536.358,E2 -536.358} C_VEL
LIN {X 0,Y 608.447,Z 579.63,A -85,B 0,C 180,E1 -537.021,E2 -537.021} C_VEL
LIN {X 0,Y 608.439,Z 582.57,A -85,B 0,C 180,E1 -538.014,E2 -538.014} C_VEL
LIN {X 0,Y 608.448,Z 583.87,A -85,B 0,C 180,E1 -538.676,E2 -538.676} C_VEL
LIN {X 0,Y 608.435,Z 584.692,A -85,B 0,C 180,E1 -539.338,E2 -539.338} C_VEL
LIN {X 0,Y 608.431,Z 584.995,A -85,B 0,C 180,E1 -540,E2 -540} C_VEL
LIN {X 0,Y 608.437,Z 584.735,A -85,B 0,C 180,E1 -540.662,E2 -540.662} C_VEL
LIN {X 0,Y 608.447,Z 583.997,A -85,B 0,C 180,E1 -541.324,E2 -541.324} C_VEL
LIN {X 0,Y 608.443,Z 582.787,A -85,B 0,C 180,E1 -541.986,E2 -541.986} C_VEL
LIN {X 0,Y 608.42,Z 579.941,A -85,B 0,C 180,E1 -542.98,E2 -542.98} C_VEL
LIN {X 0,Y 608.449,Z 577.351,A -85,B 0,C 180,E1 -543.642,E2 -543.642} C_VEL
LIN {X 0,Y 608.446,Z 572.244,A -85,B 0,C 180,E1 -544.638,E2 -544.638} C_VEL
LIN {X 0,Y 608.461,Z 566.748,A -85,B 0,C 180,E1 -545.468,E2 -545.468} C_VEL
LIN {X 0,Y 608.455,Z 559.159,A -85,B 0,C 180,E1 -546.373,E2 -546.373} C_VEL
LIN {X 0,Y 608.466,Z 550.947,A -85,B 0,C 180,E1 -547.133,E2 -547.133} C_VEL
LIN {X 0,Y 608.458,Z 543.197,A -85,B 0,C 180,E1 -547.717,E2 -547.717} C_VEL
LIN {X 0,Y 608.467,Z 535.031,A -85,B 0,C 180,E1 -548.218,E2 -548.218} C_VEL
LIN {X 0,Y 608.482,Z 531.993,A -85,B 0,C 180,E1 -548.386,E2 -548.386} C_VEL
LIN {X 0,Y 607.824,Z 528.502,A -85,B 0,C 180,E1 -548.559,E2 -548.559} C_VEL
LIN {X 0,Y 605.039,Z 523.091,A -85,B 0,C 180,E1 -548.839,E2 -548.839} C_VEL
LIN {X 0,Y 602.22,Z 517.533,A -85,B 0,C 180,E1 -549.085,E2 -549.085} C_VEL
LIN {X 0,Y 601.5,Z 513.815,A -85,B 0,C 180,E1 -549.203,E2 -549.203} C_VEL
LIN {X 0,Y 601.322,Z 506.524,A -85,B 0,C 180,E1 -549.396,E2 -549.396} C_VEL
LIN {X 0,Y 601.345,Z 501.595,A -85,B 0,C 180,E1 -552.144,E2 -552.144} C_VEL
LIN {X 0,Y 601.345,Z 496.705,A -85,B 0,C 180,E1 -554.899,E2 -554.899} C_VEL
LIN {X 0,Y 601.333,Z 491.814,A -85,B 0,C 180,E1 -557.69,E2 -557.69} C_VEL
LIN {X 0,Y 601.346,Z 486.923,A -85,B 0,C 180,E1 -560.525,E2 -560.525} C_VEL
LIN {X 0,Y 601.347,Z 482.031,A -85,B 0,C 180,E1 -563.413,E2 -563.413} C_VEL
LIN {X 0,Y 601.36,Z 477.14,A -85,B 0,C 180,E1 -566.366,E2 -566.366} C_VEL
LIN {X 0,Y 601.392,Z 475.617,A -85,B 0,C 180,E1 -567.357,E2 -567.357} C_VEL
LIN {X 0,Y 601.406,Z 480.519,A -85,B 0,C 180,E1 -569.394,E2 -569.394} C_VEL
LIN {X 0,Y 601.399,Z 488.211,A -85,B 0,C 180,E1 -572.518,E2 -572.518} C_VEL
LIN {X 0,Y 601.392,Z 494.738,A -85,B 0,C 180,E1 -575.111,E2 -575.111} C_VEL
LIN {X 0,Y 601.345,Z 501.755,A -85,B 0,C 180,E1 -577.848,E2 -577.848} C_VEL
LIN {X 0,Y 601.342,Z 508.822,A -85,B 0,C 180,E1 -580.565,E2 -580.565} C_VEL
LIN {X 0,Y 601.364,Z 515.547,A -85,B 0,C 180,E1 -583.117,E2 -583.117} C_VEL
LIN {X 0,Y 601.355,Z 523.075,A -85,B 0,C 180,E1 -585.943,E2 -585.943} C_VEL
LIN {X 0,Y 601.343,Z 525.009,A -85,B 0,C 180,E1 -586.664,E2 -586.664} C_VEL
LIN {X 0,Y 601.475,Z 537.158,A -85,B 0,C 180,E1 -586.992,E2 -586.992} C_VEL
LIN {X 0,Y 601.448,Z 546.093,A -85,B 0,C 180,E1 -587.333,E2 -587.333} C_VEL
LIN {X 0,Y 601.42,Z 555.183,A -85,B 0,C 180,E1 -587.784,E2 -587.784} C_VEL
LIN {X 0,Y 601.424,Z 564.141,A -85,B 0,C 180,E1 -588.348,E2 -588.348} C_VEL
LIN {X 0,Y 601.415,Z 572.65,A -85,B 0,C 180,E1 -589.014,E2 -589.014} C_VEL
LIN {X 0,Y 601.383,Z 580.532,A -85,B 0,C 180,E1 -589.791,E2 -589.791} C_VEL
LIN {X 0,Y 601.385,Z 587.544,A -85,B 0,C 180,E1 -590.67,E2 -590.67} C_VEL
LIN {X 0,Y 601.38,Z 591.301,A -85,B 0,C 180,E1 -591.231,E2 -591.231} C_VEL
LIN {X 0,Y 601.357,Z 596.216,A -85,B 0,C 180,E1 -592.152,E2 -592.152} C_VEL
LIN {X 0,Y 601.346,Z 599.767,A -85,B 0,C 180,E1 -593.023,E2 -593.023} C_VEL
LIN {X 0,Y 601.322,Z 602.001,A -85,B 0,C 180,E1 -593.75,E2 -593.75} C_VEL
LIN {X 0,Y 601.309,Z 603.169,A -85,B 0,C 180,E1 -594.24,E2 -594.24} C_VEL
LIN {X 0,Y 601.334,Z 604.436,A -85,B 0,C 180,E1 -595.062,E2 -595.062} C_VEL
LIN {X 0,Y 601.323,Z 604.997,A -85,B 0,C 180,E1 -596.08,E2 -596.08} C_VEL
LIN {X 0,Y 601.323,Z 604.055,A -85,B 0,C 180,E1 -597.299,E2 -597.299} C_VEL
LIN {X 0,Y 601.352,Z 601.461,A -85,B 0,C 180,E1 -598.556,E2 -598.556} C_VEL
LIN {X 0,Y 601.35,Z 598.428,A -85,B 0,C 180,E1 -599.443,E2 -599.443} C_VEL
LIN {X 0,Y 601.371,Z 593.804,A -85,B 0,C 180,E1 -600.42,E2 -600.42} C_VEL
LIN {X 0,Y 601.37,Z 588.924,A -85,B 0,C 180,E1 -601.223,E2 -601.223} C_VEL
LIN {X 0,Y 601.379,Z 583.567,A -85,B 0,C 180,E1 -601.941,E2 -601.941} C_VEL
LIN {X 0,Y 601.38,Z 576.591,A -85,B 0,C 180,E1 -602.703,E2 -602.703} C_VEL
LIN {X 0,Y 601.413,Z 568.159,A -85,B 0,C 180,E1 -603.449,E2 -603.449} C_VEL
LIN {X 0,Y 601.43,Z 558.288,A -85,B 0,C 180,E1 -604.13,E2 -604.13} C_VEL
LIN {X 0,Y 601.465,Z 549.198,A -85,B 0,C 180,E1 -604.615,E2 -604.615} C_VEL
LIN {X 0,Y 601.463,Z 540.348,A -85,B 0,C 180,E1 -604.985,E2 -604.985} C_VEL
LIN {X 0,Y 601.512,Z 531.053,A -85,B 0,C 180,E1 -605.274,E2 -605.274} C_VEL
LIN {X 0,Y 601.335,Z 525.241,A -85,B 0,C 180,E1 -605.435,E2 -605.435} C_VEL
LIN {X 0,Y 601.338,Z 518.705,A -85,B 0,C 180,E1 -608.038,E2 -608.038} C_VEL
LIN {X 0,Y 601.349,Z 511.593,A -85,B 0,C 180,E1 -610.898,E2 -610.898} C_VEL
LIN {X 0,Y 601.354,Z 504.695,A -85,B 0,C 180,E1 -613.71,E2 -613.71} C_VEL
LIN {X 0,Y 601.349,Z 498,A -85,B 0,C 180,E1 -616.482,E2 -616.482} C_VEL
LIN {X 0,Y 601.384,Z 491.494,A -85,B 0,C 180,E1 -619.223,E2 -619.223} C_VEL
LIN {X 0,Y 601.391,Z 485.181,A -85,B 0,C 180,E1 -621.938,E2 -621.938} C_VEL
LIN {X 0,Y 601.413,Z 479.05,A -85,B 0,C 180,E1 -624.635,E2 -624.635} C_VEL
LIN {X 0,Y 601.39,Z 472.831,A -85,B 0,C 180,E1 -627.32,E2 -627.32} C_VEL
LIN {X 0,Y 601.411,Z 470.386,A -85,B 0,C 180,E1 -628.326,E2 -628.326} C_VEL
LIN {X 0,Y 601.454,Z 470.381,A -85,B 0,C 180,E1 -630.669,E2 -630.669} C_VEL
LIN {X 0,Y 601.427,Z 470.382,A -85,B 0,C 180,E1 -633.349,E2 -633.349} C_VEL
LIN {X 0,Y 601.421,Z 470.383,A -85,B 0,C 180,E1 -636.037,E2 -636.037} C_VEL
LIN {X 0,Y 601.415,Z 470.387,A -85,B 0,C 180,E1 -638.738,E2 -638.738} C_VEL
LIN {X 0,Y 601.441,Z 470.381,A -85,B 0,C 180,E1 -641.458,E2 -641.458} C_VEL
LIN {X 0,Y 601.422,Z 470.383,A -85,B 0,C 180,E1 -644.205,E2 -644.205} C_VEL
LIN {X 0,Y 601.424,Z 470.385,A -85,B 0,C 180,E1 -646.986,E2 -646.986} C_VEL
LIN {X 0,Y 601.408,Z 470.385,A -85,B 0,C 180,E1 -649.809,E2 -649.809} C_VEL
LIN {X 0,Y 601.413,Z 470.385,A -85,B 0,C 180,E1 -652.683,E2 -652.683} C_VEL
LIN {X 0,Y 601.406,Z 470.385,A -85,B 0,C 180,E1 -654.878,E2 -654.878} C_VEL
LIN {X 0,Y 601.419,Z 470.385,A -85,B 0,C 180,E1 -657.867,E2 -657.867} C_VEL
LIN {X 0,Y 601.45,Z 470.382,A -85,B 0,C 180,E1 -660.162,E2 -660.162} C_VEL
LIN {X 0,Y 601.426,Z 470.383,A -85,B 0,C 180,E1 -662.716,E2 -662.716} C_VEL
LIN {X 0,Y 601.417,Z 470.384,A -85,B 0,C 180,E1 -665.115,E2 -665.115} C_VEL
LIN {X 0,Y 601.437,Z 470.382,A -85,B 0,C 180,E1 -667.418,E2 -667.418} C_VEL
LIN {X 0,Y 601.411,Z 470.384,A -85,B 0,C 180,E1 -669.995,E2 -669.995} C_VEL
LIN {X 0,Y 601.409,Z 470.385,A -85,B 0,C 180,E1 -672.67,E2 -672.67} C_VEL
LIN {X 0,Y 601.425,Z 470.386,A -85,B 0,C 180,E1 -675.482,E2 -675.482} C_VEL
LIN {X 0,Y 601.427,Z 470.382,A -85,B 0,C 180,E1 -678.406,E2 -678.406} C_VEL
LIN {X 0,Y 601.433,Z 470.381,A -85,B 0,C 180,E1 -680.875,E2 -680.875} C_VEL
LIN {X 0,Y 601.399,Z 470.387,A -85,B 0,C 180,E1 -683.417,E2 -683.417} C_VEL
LIN {X 0,Y 601.433,Z 470.385,A -85,B 0,C 180,E1 -686.064,E2 -686.064} C_VEL
LIN {X 0,Y 601.442,Z 470.383,A -85,B 0,C 180,E1 -688.541,E2 -688.541} C_VEL
LIN {X 0,Y 601.434,Z 470.381,A -85,B 0,C 180,E1 -691.373,E2 -691.373} C_VEL
LIN {X 0,Y 601.421,Z 470.385,A -85,B 0,C 180,E1 -694.13,E2 -694.13} C_VEL
LIN {X 0,Y 601.416,Z 470.386,A -85,B 0,C 180,E1 -696.589,E2 -696.589} C_VEL
LIN {X 0,Y 601.435,Z 470.381,A -85,B 0,C 180,E1 -699.478,E2 -699.478} C_VEL
LIN {X 0,Y 601.396,Z 470.387,A -85,B 0,C 180,E1 -702.312,E2 -702.312} C_VEL
LIN {X 0,Y 601.418,Z 470.383,A -85,B 0,C 180,E1 -704.409,E2 -704.409} C_VEL
LIN {X 0,Y 601.425,Z 470.384,A -85,B 0,C 180,E1 -707.172,E2 -707.172} C_VEL
LIN {X 0,Y 601.431,Z 470.383,A -85,B 0,C 180,E1 -709.905,E2 -709.905} C_VEL
LIN {X 0,Y 601.44,Z 470.38,A -85,B 0,C 180,E1 -712.615,E2 -712.615} C_VEL
LIN {X 0,Y 601.423,Z 470.383,A -85,B 0,C 180,E1 -715.308,E2 -715.308} C_VEL
LIN {X 0,Y 601.431,Z 470.385,A -85,B 0,C 180,E1 -717.991,E2 -717.991} C_VEL
LIN {X 0,Y 601.45,Z 470.38,A -85,B 0,C 180,E1 -720.669,E2 -720.669} C_VEL
LIN {X 0,Y 601.433,Z 470.381,A -85,B 0,C 180,E1 -723.349,E2 -723.349} C_VEL
LIN {X 0,Y 601.414,Z 470.386,A -85,B 0,C 180,E1 -726.037,E2 -726.037} C_VEL
LIN {X 0,Y 601.44,Z 470.383,A -85,B 0,C 180,E1 -728.738,E2 -728.738} C_VEL
LIN {X 0,Y 601.437,Z 470.381,A -85,B 0,C 180,E1 -731.458,E2 -731.458} C_VEL
LIN {X 0,Y 601.418,Z 470.384,A -85,B 0,C 180,E1 -734.205,E2 -734.205} C_VEL
LIN {X 0,Y 601.434,Z 470.384,A -85,B 0,C 180,E1 -736.986,E2 -736.986} C_VEL
LIN {X 0,Y 601.406,Z 470.385,A -85,B 0,C 180,E1 -739.809,E2 -739.809} C_VEL
LIN {X 0,Y 601.412,Z 470.387,A -85,B 0,C 180,E1 -742.683,E2 -742.683} C_VEL
LIN {X 0,Y 601.404,Z 470.386,A -85,B 0,C 180,E1 -744.878,E2 -744.878} C_VEL
LIN {X 0,Y 601.413,Z 470.386,A -85,B 0,C 180,E1 -747.363,E2 -747.363} C_VEL
LIN {X 0,Y 601.447,Z 470.38,A -85,B 0,C 180,E1 -750.163,E2 -750.163} C_VEL
LIN {X 0,Y 601.424,Z 470.382,A -85,B 0,C 180,E1 -752.716,E2 -752.716} C_VEL
LIN {X 0,Y 601.415,Z 470.384,A -85,B 0,C 180,E1 -755.115,E2 -755.115} C_VEL
LIN {X 0,Y 601.435,Z 470.381,A -85,B 0,C 180,E1 -757.419,E2 -757.419} C_VEL
LIN {X 0,Y 601.401,Z 470.385,A -85,B 0,C 180,E1 -759.996,E2 -759.996} C_VEL
LIN {X 0,Y 601.437,Z 470.383,A -85,B 0,C 180,E1 -762.668,E2 -762.668} C_VEL
LIN {X 0,Y 601.424,Z 470.384,A -85,B 0,C 180,E1 -765.482,E2 -765.482} C_VEL
LIN {X 0,Y 601.423,Z 470.383,A -85,B 0,C 180,E1 -768.407,E2 -768.407} C_VEL
LIN {X 0,Y 601.436,Z 470.382,A -85,B 0,C 180,E1 -770.876,E2 -770.876} C_VEL
LIN {X 0,Y 601.442,Z 470.382,A -85,B 0,C 180,E1 -773.734,E2 -773.734} C_VEL
LIN {X 0,Y 601.432,Z 470.383,A -85,B 0,C 180,E1 -776.064,E2 -776.064} C_VEL
LIN {X 0,Y 601.451,Z 470.576,A -85,B 0,C 180,E1 -778.81,E2 -778.81} C_VEL
LIN {X 0,Y 601.543,Z 478.058,A -85,B 0,C 180,E1 -780.946,E2 -780.946} C_VEL
LIN {X 0,Y 601.491,Z 487.752,A -85,B 0,C 180,E1 -783.641,E2 -783.641} C_VEL
LIN {X 0,Y 601.467,Z 497.264,A -85,B 0,C 180,E1 -786.227,E2 -786.227} C_VEL
LIN {X 0,Y 601.459,Z 506.776,A -85,B 0,C 180,E1 -788.763,E2 -788.763} C_VEL
LIN {X 0,Y 601.4,Z 517.647,A -85,B 0,C 180,E1 -791.608,E2 -791.608} C_VEL
LIN {X 0,Y 601.383,Z 528.518,A -85,B 0,C 180,E1 -794.408,E2 -794.408} C_VEL
LIN {X 0,Y 601.383,Z 538.03,A -85,B 0,C 180,E1 -796.828,E2 -796.828} C_VEL
LIN {X 0,Y 601.357,Z 548.901,A -85,B 0,C 180,E1 -799.564,E2 -799.564} C_VEL
LIN {X 0,Y 601.336,Z 552.978,A -85,B 0,C 180,E1 -800.583,E2 -800.583} C_VEL
LIN {X 0,Y 601.497,Z 565.244,A -85,B 0,C 180,E1 -800.882,E2 -800.882} C_VEL
LIN {X 0,Y 601.453,Z 575.544,A -85,B 0,C 180,E1 -801.263,E2 -801.263} C_VEL
LIN {X 0,Y 601.431,Z 584.241,A -85,B 0,C 180,E1 -801.686,E2 -801.686} C_VEL
LIN {X 0,Y 601.404,Z 592.548,A -85,B 0,C 180,E1 -802.193,E2 -802.193} C_VEL
LIN {X 0,Y 601.411,Z 600.405,A -85,B 0,C 180,E1 -802.784,E2 -802.784} C_VEL
LIN {X 0,Y 601.411,Z 607.599,A -85,B 0,C 180,E1 -803.443,E2 -803.443} C_VEL
LIN {X 0,Y 601.391,Z 615.194,A -85,B 0,C 180,E1 -804.3,E2 -804.3} C_VEL
LIN {X 0,Y 601.382,Z 621.029,A -85,B 0,C 180,E1 -805.14,E2 -805.14} C_VEL
LIN {X 0,Y 601.343,Z 625.632,A -85,B 0,C 180,E1 -805.979,E2 -805.979} C_VEL
LIN {X 0,Y 601.344,Z 628.623,A -85,B 0,C 180,E1 -806.65,E2 -806.65} C_VEL
LIN {X 0,Y 601.328,Z 630.933,A -85,B 0,C 180,E1 -807.321,E2 -807.321} C_VEL
LIN {X 0,Y 601.341,Z 632.679,A -85,B 0,C 180,E1 -807.991,E2 -807.991} C_VEL
LIN {X 0,Y 601.346,Z 633.935,A -85,B 0,C 180,E1 -808.661,E2 -808.661} C_VEL
LIN {X 0,Y 601.337,Z 634.714,A -85,B 0,C 180,E1 -809.331,E2 -809.331} C_VEL
LIN {X 0,Y 601.332,Z 635,A -85,B 0,C 180,E1 -810,E2 -810} C_VEL
LIN {X 0,Y 601.337,Z 634.713,A -85,B 0,C 180,E1 -810.67,E2 -810.67} C_VEL
LIN {X 0,Y 601.346,Z 633.934,A -85,B 0,C 180,E1 -811.34,E2 -811.34} C_VEL
LIN {X 0,Y 601.341,Z 632.678,A -85,B 0,C 180,E1 -812.01,E2 -812.01} C_VEL
LIN {X 0,Y 601.347,Z 629.785,A -85,B 0,C 180,E1 -813.015,E2 -813.015} C_VEL
LIN {X 0,Y 601.364,Z 627.145,A -85,B 0,C 180,E1 -813.686,E2 -813.686} C_VEL
LIN {X 0,Y 601.367,Z 621.983,A -85,B 0,C 180,E1 -814.693,E2 -814.693} C_VEL
LIN {X 0,Y 601.383,Z 616.427,A -85,B 0,C 180,E1 -815.533,E2 -815.533} C_VEL
LIN {X 0,Y 601.393,Z 609.152,A -85,B 0,C 180,E1 -816.403,E2 -816.403} C_VEL
LIN {X 0,Y 601.416,Z 601.412,A -85,B 0,C 180,E1 -817.133,E2 -817.133} C_VEL
LIN {X 0,Y 601.426,Z 593.757,A -85,B 0,C 180,E1 -817.723,E2 -817.723} C_VEL
LIN {X 0,Y 601.442,Z 585.715,A -85,B 0,C 180,E1 -818.23,E2 -818.23} C_VEL
LIN {X 0,Y 601.462,Z 577.383,A -85,B 0,C 180,E1 -818.653,E2 -818.653} C_VEL
LIN {X 0,Y 601.468,Z 568.879,A -85,B 0,C 180,E1 -818.992,E2 -818.992} C_VEL
LIN {X 0,Y 601.497,Z 559.571,A -85,B 0,C 180,E1 -819.267,E2 -819.267} C_VEL
LIN {X 0,Y 601.334,Z 553.301,A -85,B 0,C 180,E1 -819.418,E2 -819.418} C_VEL
LIN {X 0,Y 601.363,Z 543.082,A -85,B 0,C 180,E1 -822.144,E2 -822.144} C_VEL
LIN {X 0,Y 601.372,Z 532.864,A -85,B 0,C 180,E1 -824.899,E2 -824.899} C_VEL
LIN {X 0,Y 601.402,Z 522.645,A -85,B 0,C 180,E1 -827.689,E2 -827.689} C_VEL
LIN {X 0,Y 601.435,Z 512.426,A -85,B 0,C 180,E1 -830.522,E2 -830.522} C_VEL
LIN {X 0,Y 601.429,Z 503.485,A -85,B 0,C 180,E1 -833.046,E2 -833.046} C_VEL
LIN {X 0,Y 601.47,Z 494.543,A -85,B 0,C 180,E1 -835.616,E2 -835.616} C_VEL
LIN {X 0,Y 601.49,Z 485.602,A -85,B 0,C 180,E1 -838.244,E2 -838.244} C_VEL
LIN {X 0,Y 601.546,Z 476.62,A -85,B 0,C 180,E1 -840.935,E2 -840.935} C_VEL
LIN {X 0,Y 601.437,Z 470.382,A -85,B 0,C 180,E1 -842.905,E2 -842.905} C_VEL
LIN {X 0,Y 601.392,Z 470.387,A -85,B 0,C 180,E1 -845.755,E2 -845.755} C_VEL
LIN {X 0,Y 601.433,Z 470.383,A -85,B 0,C 180,E1 -848.471,E2 -848.471} C_VEL
LIN {X 0,Y 601.414,Z 470.381,A -85,B 0,C 180,E1 -850.875,E2 -850.875} C_VEL
LIN {X 0,Y 601.432,Z 470.383,A -85,B 0,C 180,E1 -853.586,E2 -853.586} C_VEL
LIN {X 0,Y 601.453,Z 470.38,A -85,B 0,C 180,E1 -856.425,E2 -856.425} C_VEL
LIN {X 0,Y 601.416,Z 470.383,A -85,B 0,C 180,E1 -859.427,E2 -859.427} C_VEL
LIN {X 0,Y 601.422,Z 470.382,A -85,B 0,C 180,E1 -861.732,E2 -861.732} C_VEL
LIN {X 0,Y 601.387,Z 470.387,A -85,B 0,C 180,E1 -864.245,E2 -864.245} C_VEL
LIN {X 0,Y 601.43,Z 470.38,A -85,B 0,C 180,E1 -866.687,E2 -866.687} C_VEL
LIN {X 0,Y 601.431,Z 470.382,A -85,B 0,C 180,E1 -867.484,E2 -867.484} C_VEL
LIN {X 0,Y 601.38,Z 471.491,A -85,B 0,C 180,E1 -868.552,E2 -868.552} C_VEL
LIN {X 0,Y 601.353,Z 475.292,A -85,B 0,C 180,E1 -871.226,E2 -871.226} C_VEL
LIN {X 0,Y 601.365,Z 479.735,A -85,B 0,C 180,E1 -874.143,E2 -874.143} C_VEL
LIN {X 0,Y 601.333,Z 483.547,A -85,B 0,C 180,E1 -876.586,E2 -876.586} C_VEL
LIN {X 0,Y 601.345,Z 488.142,A -85,B 0,C 180,E1 -879.475,E2 -879.475} C_VEL
LIN {X 0,Y 601.336,Z 492.737,A -85,B 0,C 180,E1 -882.31,E2 -882.31} C_VEL
LIN {X 0,Y 601.344,Z 497.332,A -85,B 0,C 180,E1 -885.101,E2 -885.101} C_VEL
LIN {X 0,Y 601.343,Z 501.928,A -85,B 0,C 180,E1 -887.856,E2 -887.856} C_VEL
LIN {X 0,Y 601.342,Z 506.703,A -85,B 0,C 180,E1 -890.689,E2 -890.689} C_VEL
LIN {X 0,Y 601.461,Z 518.815,A -85,B 0,C 180,E1 -891.051,E2 -891.051} C_VEL
LIN {X 0,Y 601.471,Z 526.406,A -85,B 0,C 180,E1 -891.348,E2 -891.348} C_VEL
LIN {X 0,Y 601.444,Z 534.931,A -85,B 0,C 180,E1 -891.77,E2 -891.77} C_VEL
LIN {X 0,Y 601.425,Z 543.114,A -85,B 0,C 180,E1 -892.277,E2 -892.277} C_VEL
LIN {X 0,Y 601.419,Z 550.876,A -85,B 0,C 180,E1 -892.868,E2 -892.868} C_VEL
LIN {X 0,Y 601.394,Z 558.721,A -85,B 0,C 180,E1 -893.599,E2 -893.599} C_VEL
LIN {X 0,Y 601.383,Z 566.115,A -85,B 0,C 180,E1 -894.467,E2 -894.467} C_VEL
LIN {X 0,Y 601.364,Z 571.729,A -85,B 0,C 180,E1 -895.308,E2 -895.308} C_VEL
LIN {X 0,Y 601.365,Z 576.943,A -85,B 0,C 180,E1 -896.315,E2 -896.315} C_VEL
LIN {X 0,Y 601.346,Z 579.633,A -85,B 0,C 180,E1 -896.985,E2 -896.985} C_VEL
LIN {X 0,Y 601.338,Z 582.571,A -85,B 0,C 180,E1 -897.991,E2 -897.991} C_VEL
LIN {X 0,Y 601.348,Z 583.871,A -85,B 0,C 180,E1 -898.661,E2 -898.661} C_VEL
LIN {X 0,Y 601.335,Z 584.692,A -85,B 0,C 180,E1 -899.33,E2 -899.33} C_VEL
LIN {X 0,Y 601.331,Z 584.996,A -85,B 0,C 180,E1 -900,E2 -900} C_VEL
LIN {X 0,Y 601.338,Z 584.734,A -85,B 0,C 180,E1 -900.67,E2 -900.67} C_VEL
LIN {X 0,Y 601.346,Z 583.997,A -85,B 0,C 180,E1 -901.339,E2 -901.339} C_VEL
LIN {X 0,Y 601.342,Z 582.786,A -85,B 0,C 180,E1 -902.009,E2 -902.009} C_VEL
LIN {X 0,Y 601.322,Z 579.94,A -85,B 0,C 180,E1 -903.015,E2 -903.015} C_VEL
LIN {X 0,Y 601.367,Z 577.349,A -85,B 0,C 180,E1 -903.685,E2 -903.685} C_VEL
LIN {X 0,Y 601.363,Z 572.241,A -85,B 0,C 180,E1 -904.693,E2 -904.693} C_VEL
LIN {X 0,Y 601.384,Z 566.745,A -85,B 0,C 180,E1 -905.533,E2 -905.533} C_VEL
LIN {X 0,Y 601.395,Z 558.594,A -85,B 0,C 180,E1 -906.503,E2 -906.503} C_VEL
LIN {X 0,Y 601.418,Z 550.941,A -85,B 0,C 180,E1 -907.217,E2 -907.217} C_VEL
LIN {X 0,Y 601.401,Z 543.191,A -85,B 0,C 180,E1 -907.808,E2 -907.808} C_VEL
LIN {X 0,Y 601.439,Z 535.024,A -85,B 0,C 180,E1 -908.314,E2 -908.314} C_VEL
LIN {X 0,Y 601.457,Z 524.658,A -85,B 0,C 180,E1 -908.822,E2 -908.822} C_VEL
LIN {X 0,Y 601.5,Z 513.815,A -85,B 0,C 180,E1 -909.203,E2 -909.203} C_VEL
LIN {X 0,Y 601.146,Z 510.947,A -85,B 0,C 180,E1 -909.339,E2 -909.339} C_VEL
LIN {X 0,Y 600.139,Z 508.112,A -85,B 0,C 180,E1 -909.62,E2 -909.62} C_VEL
LIN {X 0,Y 598.347,Z 505.604,A -85,B 0,C 180,E1 -910.098,E2 -910.098} C_VEL
LIN {X 0,Y 596.429,Z 504.405,A -85,B 0,C 180,E1 -910.662,E2 -910.662} C_VEL
LIN {X 0,Y 594.519,Z 503.05,A -85,B 0,C 180,E1 -911.476,E2 -911.476} C_VEL
LIN {X 0,Y 594.223,Z 502.301,A -85,B 0,C 180,E1 -911.891,E2 -911.891} C_VEL
LIN {X 0,Y 594.256,Z 497.926,A -85,B 0,C 180,E1 -914.38,E2 -914.38} C_VEL
LIN {X 0,Y 594.246,Z 493.035,A -85,B 0,C 180,E1 -917.198,E2 -917.198} C_VEL
LIN {X 0,Y 594.242,Z 488.144,A -85,B 0,C 180,E1 -920.058,E2 -920.058} C_VEL
LIN {X 0,Y 594.267,Z 483.685,A -85,B 0,C 180,E1 -922.712,E2 -922.712} C_VEL
LIN {X 0,Y 594.269,Z 479.585,A -85,B 0,C 180,E1 -925.198,E2 -925.198} C_VEL
LIN {X 0,Y 594.31,Z 476.269,A -85,B 0,C 180,E1 -927.273,E2 -927.273} C_VEL
LIN {X 0,Y 594.337,Z 482.265,A -85,B 0,C 180,E1 -929.778,E2 -929.778} C_VEL
LIN {X 0,Y 594.348,Z 488.031,A -85,B 0,C 180,E1 -932.148,E2 -932.148} C_VEL
LIN {X 0,Y 594.314,Z 494.074,A -85,B 0,C 180,E1 -934.584,E2 -934.584} C_VEL
LIN {X 0,Y 594.311,Z 500.397,A -85,B 0,C 180,E1 -937.092,E2 -937.092} C_VEL
LIN {X 0,Y 594.29,Z 507.24,A -85,B 0,C 180,E1 -939.764,E2 -939.764} C_VEL
LIN {X 0,Y 594.298,Z 515.244,A -85,B 0,C 180,E1 -942.845,E2 -942.845} C_VEL
LIN {X 0,Y 594.277,Z 522.896,A -85,B 0,C 180,E1 -945.753,E2 -945.753} C_VEL
LIN {X 0,Y 594.254,Z 525.005,A -85,B 0,C 180,E1 -946.55,E2 -946.55} C_VEL
LIN {X 0,Y 594.474,Z 537.443,A -85,B 0,C 180,E1 -946.895,E2 -946.895} C_VEL
LIN {X 0,Y 594.432,Z 546.257,A -85,B 0,C 180,E1 -947.236,E2 -947.236} C_VEL
LIN {X 0,Y 594.396,Z 555.44,A -85,B 0,C 180,E1 -947.7,E2 -947.7} C_VEL
LIN {X 0,Y 594.386,Z 563.452,A -85,B 0,C 180,E1 -948.207,E2 -948.207} C_VEL
LIN {X 0,Y 594.354,Z 572.14,A -85,B 0,C 180,E1 -948.887,E2 -948.887} C_VEL
LIN {X 0,Y 594.31,Z 579.865,A -85,B 0,C 180,E1 -949.643,E2 -949.643} C_VEL
LIN {X 0,Y 594.324,Z 587.058,A -85,B 0,C 180,E1 -950.535,E2 -950.535} C_VEL
LIN {X 0,Y 594.3,Z 592.052,A -85,B 0,C 180,E1 -951.306,E2 -951.306} C_VEL
LIN {X 0,Y 594.28,Z 595.977,A -85,B 0,C 180,E1 -952.051,E2 -952.051} C_VEL
LIN {X 0,Y 594.247,Z 600.641,A -85,B 0,C 180,E1 -953.244,E2 -953.244} C_VEL
LIN {X 0,Y 594.239,Z 602.062,A -85,B 0,C 180,E1 -953.747,E2 -953.747} C_VEL
LIN {X 0,Y 594.222,Z 603.945,A -85,B 0,C 180,E1 -954.694,E2 -954.694} C_VEL
LIN {X 0,Y 594.244,Z 604.949,A -85,B 0,C 180,E1 -955.881,E2 -955.881} C_VEL
LIN {X 0,Y 594.226,Z 604.339,A -85,B 0,C 180,E1 -957.111,E2 -957.111} C_VEL
LIN {X 0,Y 594.217,Z 603.237,A -85,B 0,C 180,E1 -957.843,E2 -957.843} C_VEL
LIN {X 0,Y 594.269,Z 601.299,A -85,B 0,C 180,E1 -958.643,E2 -958.643} C_VEL
LIN {X 0,Y 594.252,Z 597.518,A -85,B 0,C 180,E1 -959.694,E2 -959.694} C_VEL
LIN {X 0,Y 594.274,Z 593.049,A -85,B 0,C 180,E1 -960.607,E2 -960.607} C_VEL
LIN {X 0,Y 594.278,Z 588.024,A -85,B 0,C 180,E1 -961.416,E2 -961.416} C_VEL
LIN {X 0,Y 594.335,Z 582.374,A -85,B 0,C 180,E1 -962.155,E2 -962.155} C_VEL
LIN {X 0,Y 594.348,Z 574.269,A -85,B 0,C 180,E1 -963.014,E2 -963.014} C_VEL
LIN {X 0,Y 594.371,Z 565.117,A -85,B 0,C 180,E1 -963.766,E2 -963.766} C_VEL
LIN {X 0,Y 594.389,Z 556.345,A -85,B 0,C 180,E1 -964.338,E2 -964.338} C_VEL
LIN {X 0,Y 594.422,Z 547.24,A -85,B 0,C 180,E1 -964.809,E2 -964.809} C_VEL
LIN {X 0,Y 594.461,Z 536.449,A -85,B 0,C 180,E1 -965.231,E2 -965.231} C_VEL
LIN {X 0,Y 594.354,Z 526.355,A -85,B 0,C 180,E1 -965.506,E2 -965.506} C_VEL
LIN {X 0,Y 594.247,Z 525.242,A -85,B 0,C 180,E1 -965.547,E2 -965.547} C_VEL
LIN {X 0,Y 594.253,Z 519.745,A -85,B 0,C 180,E1 -967.762,E2 -967.762} C_VEL
LIN {X 0,Y 594.236,Z 514.38,A -85,B 0,C 180,E1 -969.941,E2 -969.941} C_VEL
LIN {X 0,Y 594.289,Z 507.405,A -85,B 0,C 180,E1 -972.803,E2 -972.803} C_VEL
LIN {X 0,Y 594.325,Z 500.093,A -85,B 0,C 180,E1 -975.852,E2 -975.852} C_VEL
LIN {X 0,Y 594.332,Z 492.791,A -85,B 0,C 180,E1 -978.956,E2 -978.956} C_VEL
LIN {X 0,Y 594.344,Z 486.149,A -85,B 0,C 180,E1 -981.842,E2 -981.842} C_VEL
LIN {X 0,Y 594.379,Z 480.011,A -85,B 0,C 180,E1 -984.572,E2 -984.572} C_VEL
LIN {X 0,Y 594.317,Z 473.572,A -85,B 0,C 180,E1 -987.288,E2 -987.288} C_VEL
LIN {X 0,Y 594.344,Z 471.268,A -85,B 0,C 180,E1 -988.221,E2 -988.221} C_VEL
LIN {X 0,Y 594.424,Z 471.257,A -85,B 0,C 180,E1 -990.677,E2 -990.677} C_VEL
LIN {X 0,Y 594.379,Z 471.26,A -85,B 0,C 180,E1 -993.389,E2 -993.389} C_VEL
LIN {X 0,Y 594.377,Z 471.261,A -85,B 0,C 180,E1 -996.108,E2 -996.108} C_VEL
LIN {X 0,Y 594.381,Z 471.263,A -85,B 0,C 180,E1 -998.842,E2 -998.842} C_VEL
LIN {X 0,Y 594.398,Z 471.258,A -85,B 0,C 180,E1 -1001.595,E2 -1001.595} C_VEL
LIN {X 0,Y 594.391,Z 471.259,A -85,B 0,C 180,E1 -1004.377,E2 -1004.377} C_VEL
LIN {X 0,Y 594.387,Z 471.262,A -85,B 0,C 180,E1 -1007.193,E2 -1007.193} C_VEL
LIN {X 0,Y 594.378,Z 471.26,A -85,B 0,C 180,E1 -1010.053,E2 -1010.053} C_VEL
LIN {X 0,Y 594.366,Z 471.265,A -85,B 0,C 180,E1 -1012.967,E2 -1012.967} C_VEL
LIN {X 0,Y 594.38,Z 471.262,A -85,B 0,C 180,E1 -1015.192,E2 -1015.192} C_VEL
LIN {X 0,Y 594.386,Z 471.261,A -85,B 0,C 180,E1 -1017.526,E2 -1017.526} C_VEL
LIN {X 0,Y 594.398,Z 471.258,A -85,B 0,C 180,E1 -1020.558,E2 -1020.558} C_VEL
LIN {X 0,Y 594.379,Z 471.26,A -85,B 0,C 180,E1 -1022.95,E2 -1022.95} C_VEL
LIN {X 0,Y 594.384,Z 471.259,A -85,B 0,C 180,E1 -1025.406,E2 -1025.406} C_VEL
LIN {X 0,Y 594.39,Z 471.259,A -85,B 0,C 180,E1 -1027.94,E2 -1027.94} C_VEL
LIN {X 0,Y 594.374,Z 471.263,A -85,B 0,C 180,E1 -1030.822,E2 -1030.822} C_VEL
LIN {X 0,Y 594.382,Z 471.26,A -85,B 0,C 180,E1 -1033.841,E2 -1033.841} C_VEL
LIN {X 0,Y 594.379,Z 471.263,A -85,B 0,C 180,E1 -1036.702,E2 -1036.702} C_VEL
LIN {X 0,Y 594.39,Z 471.259,A -85,B 0,C 180,E1 -1039.435,E2 -1039.435} C_VEL
LIN {X 0,Y 594.389,Z 471.261,A -85,B 0,C 180,E1 -1042.391,E2 -1042.391} C_VEL
LIN {X 0,Y 594.381,Z 471.26,A -85,B 0,C 180,E1 -1045.42,E2 -1045.42} C_VEL
LIN {X 0,Y 594.393,Z 471.261,A -85,B 0,C 180,E1 -1048.354,E2 -1048.354} C_VEL
LIN {X 0,Y 594.382,Z 471.261,A -85,B 0,C 180,E1 -1051.042,E2 -1051.042} C_VEL
LIN {X 0,Y 594.394,Z 471.259,A -85,B 0,C 180,E1 -1053.975,E2 -1053.975} C_VEL
LIN {X 0,Y 594.386,Z 471.26,A -85,B 0,C 180,E1 -1056.296,E2 -1056.296} C_VEL
LIN {X 0,Y 594.407,Z 471.259,A -85,B 0,C 180,E1 -1059.224,E2 -1059.224} C_VEL
LIN {X 0,Y 594.353,Z 471.263,A -85,B 0,C 180,E1 -1062.095,E2 -1062.095} C_VEL
LIN {X 0,Y 594.371,Z 471.261,A -85,B 0,C 180,E1 -1064.219,E2 -1064.219} C_VEL
LIN {X 0,Y 594.371,Z 471.262,A -85,B 0,C 180,E1 -1067.017,E2 -1067.017} C_VEL
LIN {X 0,Y 594.391,Z 471.261,A -85,B 0,C 180,E1 -1069.784,E2 -1069.784} C_VEL
LIN {X 0,Y 594.393,Z 471.258,A -85,B 0,C 180,E1 -1072.527,E2 -1072.527} C_VEL
LIN {X 0,Y 594.392,Z 471.259,A -85,B 0,C 180,E1 -1075.252,E2 -1075.252} C_VEL
LIN {X 0,Y 594.401,Z 471.261,A -85,B 0,C 180,E1 -1077.967,E2 -1077.967} C_VEL
LIN {X 0,Y 594.421,Z 471.255,A -85,B 0,C 180,E1 -1080.677,E2 -1080.677} C_VEL
LIN {X 0,Y 594.384,Z 471.259,A -85,B 0,C 180,E1 -1083.389,E2 -1083.389} C_VEL
LIN {X 0,Y 594.37,Z 471.264,A -85,B 0,C 180,E1 -1086.109,E2 -1086.109} C_VEL
LIN {X 0,Y 594.4,Z 471.259,A -85,B 0,C 180,E1 -1088.842,E2 -1088.842} C_VEL
LIN {X 0,Y 594.395,Z 471.258,A -85,B 0,C 180,E1 -1091.596,E2 -1091.596} C_VEL
LIN {X 0,Y 594.388,Z 471.261,A -85,B 0,C 180,E1 -1094.377,E2 -1094.377} C_VEL
LIN {X 0,Y 594.392,Z 471.259,A -85,B 0,C 180,E1 -1097.193,E2 -1097.193} C_VEL
LIN {X 0,Y 594.375,Z 471.261,A -85,B 0,C 180,E1 -1100.054,E2 -1100.054} C_VEL
LIN {X 0,Y 594.365,Z 471.264,A -85,B 0,C 180,E1 -1102.967,E2 -1102.967} C_VEL
LIN {X 0,Y 594.375,Z 471.264,A -85,B 0,C 180,E1 -1105.193,E2 -1105.193} C_VEL
LIN {X 0,Y 594.383,Z 471.263,A -85,B 0,C 180,E1 -1107.527,E2 -1107.527} C_VEL
LIN {X 0,Y 594.399,Z 471.257,A -85,B 0,C 180,E1 -1110.331,E2 -1110.331} C_VEL
LIN {X 0,Y 594.378,Z 471.26,A -85,B 0,C 180,E1 -1112.95,E2 -1112.95} C_VEL
LIN {X 0,Y 594.383,Z 471.26,A -85,B 0,C 180,E1 -1115.407,E2 -1115.407} C_VEL
LIN {X 0,Y 594.388,Z 471.261,A -85,B 0,C 180,E1 -1117.941,E2 -1117.941} C_VEL
LIN {X 0,Y 594.38,Z 471.261,A -85,B 0,C 180,E1 -1120.823,E2 -1120.823} C_VEL
LIN {X 0,Y 594.385,Z 471.26,A -85,B 0,C 180,E1 -1123.298,E2 -1123.298} C_VEL
LIN {X 0,Y 594.366,Z 471.263,A -85,B 0,C 180,E1 -1126.161,E2 -1126.161} C_VEL
LIN {X 0,Y 594.39,Z 471.259,A -85,B 0,C 180,E1 -1129.177,E2 -1129.177} C_VEL
LIN {X 0,Y 594.385,Z 471.261,A -85,B 0,C 180,E1 -1132.06,E2 -1132.06} C_VEL
LIN {X 0,Y 594.386,Z 471.263,A -85,B 0,C 180,E1 -1134.672,E2 -1134.672} C_VEL
LIN {X 0,Y 594.377,Z 471.264,A -85,B 0,C 180,E1 -1137.089,E2 -1137.089} C_VEL
LIN {X 0,Y 594.411,Z 471.449,A -85,B 0,C 180,E1 -1138.653,E2 -1138.653} C_VEL
LIN {X 0,Y 594.557,Z 476.849,A -85,B 0,C 180,E1 -1140.234,E2 -1140.234} C_VEL
LIN {X 0,Y 594.522,Z 486.393,A -85,B 0,C 180,E1 -1142.928,E2 -1142.928} C_VEL
LIN {X 0,Y 594.457,Z 497.264,A -85,B 0,C 180,E1 -1145.929,E2 -1145.929} C_VEL
LIN {X 0,Y 594.412,Z 508.019,A -85,B 0,C 180,E1 -1148.831,E2 -1148.831} C_VEL
LIN {X 0,Y 594.376,Z 517.647,A -85,B 0,C 180,E1 -1151.383,E2 -1151.383} C_VEL
LIN {X 0,Y 594.327,Z 528.518,A -85,B 0,C 180,E1 -1154.218,E2 -1154.218} C_VEL
LIN {X 0,Y 594.307,Z 538.03,A -85,B 0,C 180,E1 -1156.668,E2 -1156.668} C_VEL
LIN {X 0,Y 594.284,Z 548.901,A -85,B 0,C 180,E1 -1159.438,E2 -1159.438} C_VEL
LIN {X 0,Y 594.265,Z 552.978,A -85,B 0,C 180,E1 -1160.47,E2 -1160.47} C_VEL
LIN {X 0,Y 594.509,Z 563.748,A -85,B 0,C 180,E1 -1160.731,E2 -1160.731} C_VEL
LIN {X 0,Y 594.443,Z 575.543,A -85,B 0,C 180,E1 -1161.159,E2 -1161.159} C_VEL
LIN {X 0,Y 594.406,Z 584.243,A -85,B 0,C 180,E1 -1161.587,E2 -1161.587} C_VEL
LIN {X 0,Y 594.373,Z 592.55,A -85,B 0,C 180,E1 -1162.1,E2 -1162.1} C_VEL
LIN {X 0,Y 594.351,Z 600.406,A -85,B 0,C 180,E1 -1162.697,E2 -1162.697} C_VEL
LIN {X 0,Y 594.342,Z 607.516,A -85,B 0,C 180,E1 -1163.357,E2 -1163.357} C_VEL
LIN {X 0,Y 594.318,Z 615.193,A -85,B 0,C 180,E1 -1164.232,E2 -1164.232} C_VEL
LIN {X 0,Y 594.291,Z 621.03,A -85,B 0,C 180,E1 -1165.082,E2 -1165.082} C_VEL
LIN {X 0,Y 594.26,Z 625.633,A -85,B 0,C 180,E1 -1165.931,E2 -1165.931} C_VEL
LIN {X 0,Y 594.267,Z 628.623,A -85,B 0,C 180,E1 -1166.61,E2 -1166.61} C_VEL
LIN {X 0,Y 594.231,Z 630.933,A -85,B 0,C 180,E1 -1167.289,E2 -1167.289} C_VEL
LIN {X 0,Y 594.24,Z 632.68,A -85,B 0,C 180,E1 -1167.967,E2 -1167.967} C_VEL
LIN {X 0,Y 594.246,Z 633.935,A -85,B 0,C 180,E1 -1168.645,E2 -1168.645} C_VEL
LIN {X 0,Y 594.237,Z 634.713,A -85,B 0,C 180,E1 -1169.323,E2 -1169.323} C_VEL
LIN {X 0,Y 594.233,Z 635,A -85,B 0,C 180,E1 -1170,E2 -1170} C_VEL
LIN {X 0,Y 594.237,Z 634.713,A -85,B 0,C 180,E1 -1170.678,E2 -1170.678} C_VEL
LIN {X 0,Y 594.246,Z 633.934,A -85,B 0,C 180,E1 -1171.356,E2 -1171.356} C_VEL
LIN {X 0,Y 594.24,Z 632.678,A -85,B 0,C 180,E1 -1172.034,E2 -1172.034} C_VEL
LIN {X 0,Y 594.249,Z 629.786,A -85,B 0,C 180,E1 -1173.051,E2 -1173.051} C_VEL
LIN {X 0,Y 594.285,Z 627.145,A -85,B 0,C 180,E1 -1173.73,E2 -1173.73} C_VEL
LIN {X 0,Y 594.277,Z 621.983,A -85,B 0,C 180,E1 -1174.749,E2 -1174.749} C_VEL
LIN {X 0,Y 594.309,Z 616.428,A -85,B 0,C 180,E1 -1175.599,E2 -1175.599} C_VEL
LIN {X 0,Y 594.344,Z 609.151,A -85,B 0,C 180,E1 -1176.479,E2 -1176.479} C_VEL
LIN {X 0,Y 594.356,Z 601.413,A -85,B 0,C 180,E1 -1177.218,E2 -1177.218} C_VEL
LIN {X 0,Y 594.361,Z 593.759,A -85,B 0,C 180,E1 -1177.816,E2 -1177.816} C_VEL
LIN {X 0,Y 594.418,Z 585.717,A -85,B 0,C 180,E1 -1178.328,E2 -1178.328} C_VEL
LIN {X 0,Y 594.427,Z 577.386,A -85,B 0,C 180,E1 -1178.756,E2 -1178.756} C_VEL
LIN {X 0,Y 594.461,Z 568.881,A -85,B 0,C 180,E1 -1179.098,E2 -1179.098} C_VEL
LIN {X 0,Y 594.482,Z 558.741,A -85,B 0,C 180,E1 -1179.398,E2 -1179.398} C_VEL
LIN {X 0,Y 594.258,Z 553.301,A -85,B 0,C 180,E1 -1179.531,E2 -1179.531} C_VEL
LIN {X 0,Y 594.295,Z 543.082,A -85,B 0,C 180,E1 -1182.291,E2 -1182.291} C_VEL
LIN {X 0,Y 594.304,Z 532.864,A -85,B 0,C 180,E1 -1185.08,E2 -1185.08} C_VEL
LIN {X 0,Y 594.362,Z 522.645,A -85,B 0,C 180,E1 -1187.905,E2 -1187.905} C_VEL
LIN {X 0,Y 594.391,Z 512.426,A -85,B 0,C 180,E1 -1190.776,E2 -1190.776} C_VEL
LIN {X 0,Y 594.421,Z 503.485,A -85,B 0,C 180,E1 -1193.334,E2 -1193.334} C_VEL
LIN {X 0,Y 594.459,Z 494.216,A -85,B 0,C 180,E1 -1196.037,E2 -1196.037} C_VEL
LIN {X 0,Y 594.499,Z 485.622,A -85,B 0,C 180,E1 -1198.6,E2 -1198.6} C_VEL
LIN {X 0,Y 594.562,Z 476.591,A -85,B 0,C 180,E1 -1201.339,E2 -1201.339} C_VEL
LIN {X 0,Y 594.396,Z 471.26,A -85,B 0,C 180,E1 -1203.076,E2 -1203.076} C_VEL
LIN {X 0,Y 594.36,Z 471.266,A -85,B 0,C 180,E1 -1205.409,E2 -1205.409} C_VEL
LIN {X 0,Y 594.387,Z 471.257,A -85,B 0,C 180,E1 -1207.941,E2 -1207.941} C_VEL
LIN {X 0,Y 594.378,Z 471.258,A -85,B 0,C 180,E1 -1210.822,E2 -1210.822} C_VEL
LIN {X 0,Y 594.369,Z 471.264,A -85,B 0,C 180,E1 -1213.3,E2 -1213.3} C_VEL
LIN {X 0,Y 594.385,Z 471.258,A -85,B 0,C 180,E1 -1216.159,E2 -1216.159} C_VEL
LIN {X 0,Y 594.379,Z 471.258,A -85,B 0,C 180,E1 -1219.178,E2 -1219.178} C_VEL
LIN {X 0,Y 594.388,Z 471.256,A -85,B 0,C 180,E1 -1222.06,E2 -1222.06} C_VEL
LIN {X 0,Y 594.352,Z 471.266,A -85,B 0,C 180,E1 -1224.677,E2 -1224.677} C_VEL
LIN {X 0,Y 594.382,Z 471.257,A -85,B 0,C 180,E1 -1227.089,E2 -1227.089} C_VEL
LIN {X 0,Y 594.33,Z 471.27,A -85,B 0,C 180,E1 -1227.851,E2 -1227.851} C_VEL
LIN {X 0,Y 594.289,Z 474.552,A -85,B 0,C 180,E1 -1230.219,E2 -1230.219} C_VEL
LIN {X 0,Y 594.267,Z 477.805,A -85,B 0,C 180,E1 -1232.534,E2 -1232.534} C_VEL
LIN {X 0,Y 594.256,Z 481.251,A -85,B 0,C 180,E1 -1234.802,E2 -1234.802} C_VEL
LIN {X 0,Y 594.261,Z 485.846,A -85,B 0,C 180,E1 -1237.763,E2 -1237.763} C_VEL
LIN {X 0,Y 594.24,Z 489.292,A -85,B 0,C 180,E1 -1239.942,E2 -1239.942} C_VEL
LIN {X 0,Y 594.247,Z 493.887,A -85,B 0,C 180,E1 -1242.802,E2 -1242.802} C_VEL
LIN {X 0,Y 594.255,Z 498.482,A -85,B 0,C 180,E1 -1245.62,E2 -1245.62} C_VEL
LIN {X 0,Y 594.229,Z 503.078,A -85,B 0,C 180,E1 -1248.401,E2 -1248.401} C_VEL
LIN {X 0,Y 594.231,Z 506.704,A -85,B 0,C 180,E1 -1250.577,E2 -1250.577} C_VEL
LIN {X 0,Y 594.514,Z 512.826,A -85,B 0,C 180,E1 -1250.753,E2 -1250.753} C_VEL
LIN {X 0,Y 594.446,Z 524.553,A -85,B 0,C 180,E1 -1251.159,E2 -1251.159} C_VEL
LIN {X 0,Y 594.424,Z 534.943,A -85,B 0,C 180,E1 -1251.672,E2 -1251.672} C_VEL
LIN {X 0,Y 594.361,Z 543.124,A -85,B 0,C 180,E1 -1252.185,E2 -1252.185} C_VEL
LIN {X 0,Y 594.361,Z 550.883,A -85,B 0,C 180,E1 -1252.783,E2 -1252.783} C_VEL
LIN {X 0,Y 594.345,Z 558.726,A -85,B 0,C 180,E1 -1253.523,E2 -1253.523} C_VEL
LIN {X 0,Y 594.309,Z 566.119,A -85,B 0,C 180,E1 -1254.401,E2 -1254.401} C_VEL
LIN {X 0,Y 594.274,Z 571.732,A -85,B 0,C 180,E1 -1255.251,E2 -1255.251} C_VEL
LIN {X 0,Y 594.286,Z 576.946,A -85,B 0,C 180,E1 -1256.271,E2 -1256.271} C_VEL
LIN {X 0,Y 594.249,Z 579.635,A -85,B 0,C 180,E1 -1256.949,E2 -1256.949} C_VEL
LIN {X 0,Y 594.238,Z 582.573,A -85,B 0,C 180,E1 -1257.967,E2 -1257.967} C_VEL
LIN {X 0,Y 594.248,Z 583.872,A -85,B 0,C 180,E1 -1258.645,E2 -1258.645} C_VEL
LIN {X 0,Y 594.236,Z 584.692,A -85,B 0,C 180,E1 -1259.322,E2 -1259.322} C_VEL
LIN {X 0,Y 594.232,Z 584.996,A -85,B 0,C 180,E1 -1260,E2 -1260} C_VEL
LIN {X 0,Y 594.238,Z 584.734,A -85,B 0,C 180,E1 -1260.678,E2 -1260.678} C_VEL
LIN {X 0,Y 594.246,Z 583.997,A -85,B 0,C 180,E1 -1261.355,E2 -1261.355} C_VEL
LIN {X 0,Y 594.241,Z 582.785,A -85,B 0,C 180,E1 -1262.033,E2 -1262.033} C_VEL
LIN {X 0,Y 594.229,Z 579.939,A -85,B 0,C 180,E1 -1263.051,E2 -1263.051} C_VEL
LIN {X 0,Y 594.288,Z 577.347,A -85,B 0,C 180,E1 -1263.729,E2 -1263.729} C_VEL
LIN {X 0,Y 594.266,Z 572.239,A -85,B 0,C 180,E1 -1264.749,E2 -1264.749} C_VEL
LIN {X 0,Y 594.31,Z 566.742,A -85,B 0,C 180,E1 -1265.599,E2 -1265.599} C_VEL
LIN {X 0,Y 594.334,Z 558.789,A -85,B 0,C 180,E1 -1266.56,E2 -1266.56} C_VEL
LIN {X 0,Y 594.359,Z 550.935,A -85,B 0,C 180,E1 -1267.303,E2 -1267.303} C_VEL
LIN {X 0,Y 594.367,Z 543.185,A -85,B 0,C 180,E1 -1267.901,E2 -1267.901} C_VEL
LIN {X 0,Y 594.414,Z 535.017,A -85,B 0,C 180,E1 -1268.413,E2 -1268.413} C_VEL
LIN {X 0,Y 594.458,Z 524.644,A -85,B 0,C 180,E1 -1268.927,E2 -1268.927} C_VEL
LIN {X 0,Y 594.492,Z 512.983,A -85,B 0,C 180,E1 -1269.334,E2 -1269.334} C_VEL
LIN {X 0,Y 594.23,Z 506.523,A -85,B 0,C 180,E1 -1269.509,E2 -1269.509} C_VEL
LIN {X 0,Y 594.223,Z 502.301,A -85,B 0,C 180,E1 -1271.891,E2 -1271.891} C_VEL
LIN {X 0,Y 593.567,Z 501.34,A -85,B 0,C 180,E1 -1272.45,E2 -1272.45} C_VEL
LIN {X 0,Y 590.716,Z 499.86,A -85,B 0,C 180,E1 -1273.358,E2 -1273.358} C_VEL
LIN {X 0,Y 588.297,Z 498.689,A -85,B 0,C 180,E1 -1274.088,E2 -1274.088} C_VEL
LIN {X 0,Y 587.253,Z 497.761,A -85,B 0,C 180,E1 -1274.651,E2 -1274.651} C_VEL
LIN {X 0,Y 587.165,Z 497.436,A -85,B 0,C 180,E1 -1274.842,E2 -1274.842} C_VEL
LIN {X 0,Y 587.143,Z 493.034,A -85,B 0,C 180,E1 -1277.412,E2 -1277.412} C_VEL
LIN {X 0,Y 587.154,Z 489.366,A -85,B 0,C 180,E1 -1279.582,E2 -1279.582} C_VEL
LIN {X 0,Y 587.175,Z 485.698,A -85,B 0,C 180,E1 -1281.78,E2 -1281.78} C_VEL
LIN {X 0,Y 587.198,Z 481.162,A -85,B 0,C 180,E1 -1284.546,E2 -1284.546} C_VEL
LIN {X 0,Y 587.255,Z 476.87,A -85,B 0,C 180,E1 -1287.288,E2 -1287.288} C_VEL
LIN {X 0,Y 587.288,Z 482.133,A -85,B 0,C 180,E1 -1289.383,E2 -1289.383} C_VEL
LIN {X 0,Y 587.285,Z 489.828,A -85,B 0,C 180,E1 -1292.582,E2 -1292.582} C_VEL
LIN {X 0,Y 587.235,Z 495.927,A -85,B 0,C 180,E1 -1295.062,E2 -1295.062} C_VEL
LIN {X 0,Y 587.214,Z 502.831,A -85,B 0,C 180,E1 -1297.822,E2 -1297.822} C_VEL
LIN {X 0,Y 587.203,Z 509.03,A -85,B 0,C 180,E1 -1300.264,E2 -1300.264} C_VEL
LIN {X 0,Y 587.216,Z 516.343,A -85,B 0,C 180,E1 -1303.107,E2 -1303.107} C_VEL
LIN {X 0,Y 587.189,Z 523.609,A -85,B 0,C 180,E1 -1305.901,E2 -1305.901} C_VEL
LIN {X 0,Y 587.171,Z 525.022,A -85,B 0,C 180,E1 -1306.441,E2 -1306.441} C_VEL
LIN {X 0,Y 587.508,Z 532.14,A -85,B 0,C 180,E1 -1306.622,E2 -1306.622} C_VEL
LIN {X 0,Y 587.443,Z 543.452,A -85,B 0,C 180,E1 -1307.005,E2 -1307.005} C_VEL
LIN {X 0,Y 587.392,Z 553.188,A -85,B 0,C 180,E1 -1307.468,E2 -1307.468} C_VEL
LIN {X 0,Y 587.355,Z 562.479,A -85,B 0,C 180,E1 -1308.043,E2 -1308.043} C_VEL
LIN {X 0,Y 587.303,Z 571.275,A -85,B 0,C 180,E1 -1308.726,E2 -1308.726} C_VEL
LIN {X 0,Y 587.237,Z 579.39,A -85,B 0,C 180,E1 -1309.514,E2 -1309.514} C_VEL
LIN {X 0,Y 587.243,Z 587.092,A -85,B 0,C 180,E1 -1310.472,E2 -1310.472} C_VEL
LIN {X 0,Y 587.229,Z 592.309,A -85,B 0,C 180,E1 -1311.294,E2 -1311.294} C_VEL
LIN {X 0,Y 587.165,Z 596.782,A -85,B 0,C 180,E1 -1312.184,E2 -1312.184} C_VEL
LIN {X 0,Y 587.143,Z 601.008,A -85,B 0,C 180,E1 -1313.319,E2 -1313.319} C_VEL
LIN {X 0,Y 587.134,Z 603.673,A -85,B 0,C 180,E1 -1314.485,E2 -1314.485} C_VEL
LIN {X 0,Y 587.141,Z 604.898,A -85,B 0,C 180,E1 -1315.765,E2 -1315.765} C_VEL
LIN {X 0,Y 587.12,Z 604.595,A -85,B 0,C 180,E1 -1316.921,E2 -1316.921} C_VEL
LIN {X 0,Y 587.149,Z 602.419,A -85,B 0,C 180,E1 -1318.219,E2 -1318.219} C_VEL
LIN {X 0,Y 587.162,Z 600.166,A -85,B 0,C 180,E1 -1319.023,E2 -1319.023} C_VEL
LIN {X 0,Y 587.183,Z 597.158,A -85,B 0,C 180,E1 -1319.821,E2 -1319.821} C_VEL
LIN {X 0,Y 587.194,Z 593.338,A -85,B 0,C 180,E1 -1320.612,E2 -1320.612} C_VEL
LIN {X 0,Y 587.19,Z 588.615,A -85,B 0,C 180,E1 -1321.396,E2 -1321.396} C_VEL
LIN {X 0,Y 587.274,Z 581.612,A -85,B 0,C 180,E1 -1322.322,E2 -1322.322} C_VEL
LIN {X 0,Y 587.273,Z 572.721,A -85,B 0,C 180,E1 -1323.239,E2 -1323.239} C_VEL
LIN {X 0,Y 587.335,Z 564.389,A -85,B 0,C 180,E1 -1323.912,E2 -1323.912} C_VEL
LIN {X 0,Y 587.366,Z 555.56,A -85,B 0,C 180,E1 -1324.485,E2 -1324.485} C_VEL
LIN {X 0,Y 587.407,Z 545.254,A -85,B 0,C 180,E1 -1325.007,E2 -1325.007} C_VEL
LIN {X 0,Y 587.528,Z 533.555,A -85,B 0,C 180,E1 -1325.429,E2 -1325.429} C_VEL
LIN {X 0,Y 587.232,Z 526.219,A -85,B 0,C 180,E1 -1325.624,E2 -1325.624} C_VEL
LIN {X 0,Y 587.154,Z 525.247,A -85,B 0,C 180,E1 -1325.661,E2 -1325.661} C_VEL
LIN {X 0,Y 587.142,Z 518.982,A -85,B 0,C 180,E1 -1328.218,E2 -1328.218} C_VEL
LIN {X 0,Y 587.208,Z 511.879,A -85,B 0,C 180,E1 -1331.146,E2 -1331.146} C_VEL
LIN {X 0,Y 587.218,Z 505,A -85,B 0,C 180,E1 -1334.022,E2 -1334.022} C_VEL
LIN {X 0,Y 587.202,Z 498.331,A -85,B 0,C 180,E1 -1336.855,E2 -1336.855} C_VEL
LIN {X 0,Y 587.273,Z 491.849,A -85,B 0,C 180,E1 -1339.659,E2 -1339.659} C_VEL
LIN {X 0,Y 587.273,Z 485.568,A -85,B 0,C 180,E1 -1342.435,E2 -1342.435} C_VEL
LIN {X 0,Y 587.3,Z 479.159,A -85,B 0,C 180,E1 -1345.195,E2 -1345.195} C_VEL
LIN {X 0,Y 587.321,Z 472.143,A -85,B 0,C 180,E1 -1348.2,E2 -1348.2} C_VEL
LIN {X 0,Y 587.395,Z 472.132,A -85,B 0,C 180,E1 -1350.685,E2 -1350.685} C_VEL
LIN {X 0,Y 587.33,Z 472.138,A -85,B 0,C 180,E1 -1353.43,E2 -1353.43} C_VEL
LIN {X 0,Y 587.367,Z 472.135,A -85,B 0,C 180,E1 -1355.493,E2 -1355.493} C_VEL
LIN {X 0,Y 587.369,Z 472.133,A -85,B 0,C 180,E1 -1358.255,E2 -1358.255} C_VEL
LIN {X 0,Y 587.35,Z 472.139,A -85,B 0,C 180,E1 -1361.133,E2 -1361.133} C_VEL
LIN {X 0,Y 587.367,Z 472.134,A -85,B 0,C 180,E1 -1364.26,E2 -1364.26} C_VEL
LIN {X 0,Y 587.357,Z 472.135,A -85,B 0,C 180,E1 -1367.405,E2 -1367.405} C_VEL
LIN {X 0,Y 587.333,Z 472.139,A -85,B 0,C 180,E1 -1370.304,E2 -1370.304} C_VEL
LIN {X 0,Y 587.325,Z 472.14,A -85,B 0,C 180,E1 -1373.258,E2 -1373.258} C_VEL
LIN {X 0,Y 587.34,Z 472.139,A -85,B 0,C 180,E1 -1375.516,E2 -1375.516} C_VEL
LIN {X 0,Y 587.349,Z 472.139,A -85,B 0,C 180,E1 -1377.817,E2 -1377.817} C_VEL
LIN {X 0,Y 587.353,Z 472.135,A -85,B 0,C 180,E1 -1380.512,E2 -1380.512} C_VEL
LIN {X 0,Y 587.336,Z 472.139,A -85,B 0,C 180,E1 -1383.396,E2 -1383.396} C_VEL
LIN {X 0,Y 587.357,Z 472.137,A -85,B 0,C 180,E1 -1385.895,E2 -1385.895} C_VEL
LIN {X 0,Y 587.334,Z 472.14,A -85,B 0,C 180,E1 -1388.479,E2 -1388.479} C_VEL
LIN {X 0,Y 587.334,Z 472.138,A -85,B 0,C 180,E1 -1391.157,E2 -1391.157} C_VEL
LIN {X 0,Y 587.334,Z 472.14,A -85,B 0,C 180,E1 -1394.114,E2 -1394.114} C_VEL
LIN {X 0,Y 587.321,Z 472.139,A -85,B 0,C 180,E1 -1396.994,E2 -1396.994} C_VEL
LIN {X 0,Y 587.329,Z 472.139,A -85,B 0,C 180,E1 -1399.747,E2 -1399.747} C_VEL
LIN {X 0,Y 587.345,Z 472.139,A -85,B 0,C 180,E1 -1402.392,E2 -1402.392} C_VEL
LIN {X 0,Y 587.362,Z 472.135,A -85,B 0,C 180,E1 -1405.78,E2 -1405.78} C_VEL
LIN {X 0,Y 587.355,Z 472.137,A -85,B 0,C 180,E1 -1408.232,E2 -1408.232} C_VEL
LIN {X 0,Y 587.348,Z 472.139,A -85,B 0,C 180,E1 -1410.866,E2 -1410.866} C_VEL
LIN {X 0,Y 587.363,Z 472.134,A -85,B 0,C 180,E1 -1413.818,E2 -1413.818} C_VEL
LIN {X 0,Y 587.334,Z 472.138,A -85,B 0,C 180,E1 -1415.993,E2 -1415.993} C_VEL
LIN {X 0,Y 587.347,Z 472.139,A -85,B 0,C 180,E1 -1418.963,E2 -1418.963} C_VEL
LIN {X 0,Y 587.351,Z 472.136,A -85,B 0,C 180,E1 -1421.151,E2 -1421.151} C_VEL
LIN {X 0,Y 587.328,Z 472.14,A -85,B 0,C 180,E1 -1424.025,E2 -1424.025} C_VEL
LIN {X 0,Y 587.36,Z 472.138,A -85,B 0,C 180,E1 -1426.154,E2 -1426.154} C_VEL
LIN {X 0,Y 587.341,Z 472.137,A -85,B 0,C 180,E1 -1428.962,E2 -1428.962} C_VEL
LIN {X 0,Y 587.371,Z 472.134,A -85,B 0,C 180,E1 -1431.745,E2 -1431.745} C_VEL
LIN {X 0,Y 587.356,Z 472.137,A -85,B 0,C 180,E1 -1434.507,E2 -1434.507} C_VEL
LIN {X 0,Y 587.379,Z 472.132,A -85,B 0,C 180,E1 -1437.257,E2 -1437.257} C_VEL
LIN {X 0,Y 587.382,Z 472.133,A -85,B 0,C 180,E1 -1440,E2 -1440} C_VEL
LIN {X 0,Y 587.378,Z 472.135,A -85,B 0,C 180,E1 -1442.743,E2 -1442.743} C_VEL
LIN {X 0,Y 587.362,Z 472.134,A -85,B 0,C 180,E1 -1445.493,E2 -1445.493} C_VEL
LIN {X 0,Y 587.368,Z 472.134,A -85,B 0,C 180,E1 -1448.255,E2 -1448.255} C_VEL
LIN {X 0,Y 587.346,Z 472.138,A -85,B 0,C 180,E1 -1451.134,E2 -1451.134} C_VEL
LIN {X 0,Y 587.363,Z 472.135,A -85,B 0,C 180,E1 -1454.261,E2 -1454.261} C_VEL
LIN {X 0,Y 587.359,Z 472.135,A -85,B 0,C 180,E1 -1457.406,E2 -1457.406} C_VEL
LIN {X 0,Y 587.33,Z 472.141,A -85,B 0,C 180,E1 -1460.305,E2 -1460.305} C_VEL
LIN {X 0,Y 587.324,Z 472.139,A -85,B 0,C 180,E1 -1463.259,E2 -1463.259} C_VEL
LIN {X 0,Y 587.333,Z 472.138,A -85,B 0,C 180,E1 -1465.517,E2 -1465.517} C_VEL
LIN {X 0,Y 587.346,Z 472.137,A -85,B 0,C 180,E1 -1467.818,E2 -1467.818} C_VEL
LIN {X 0,Y 587.349,Z 472.135,A -85,B 0,C 180,E1 -1470.513,E2 -1470.513} C_VEL
LIN {X 0,Y 587.334,Z 472.141,A -85,B 0,C 180,E1 -1473.397,E2 -1473.397} C_VEL
LIN {X 0,Y 587.356,Z 472.137,A -85,B 0,C 180,E1 -1475.895,E2 -1475.895} C_VEL
LIN {X 0,Y 587.329,Z 472.139,A -85,B 0,C 180,E1 -1478.479,E2 -1478.479} C_VEL
LIN {X 0,Y 587.337,Z 472.137,A -85,B 0,C 180,E1 -1481.157,E2 -1481.157} C_VEL
LIN {X 0,Y 587.333,Z 472.14,A -85,B 0,C 180,E1 -1484.115,E2 -1484.115} C_VEL
LIN {X 0,Y 587.314,Z 472.14,A -85,B 0,C 180,E1 -1486.994,E2 -1486.994} C_VEL
LIN {X 0,Y 587.329,Z 472.14,A -85,B 0,C 180,E1 -1489.747,E2 -1489.747} C_VEL
LIN {X 0,Y 587.343,Z 472.139,A -85,B 0,C 180,E1 -1492.393,E2 -1492.393} C_VEL
LIN {X 0,Y 587.351,Z 472.137,A -85,B 0,C 180,E1 -1494.947,E2 -1494.947} C_VEL
LIN {X 0,Y 587.336,Z 472.139,A -85,B 0,C 180,E1 -1497.421,E2 -1497.421} C_VEL
LIN {X 0,Y 587.401,Z 472.301,A -85,B 0,C 180,E1 -1498.487,E2 -1498.487} C_VEL
LIN {X 0,Y 587.588,Z 476.839,A -85,B 0,C 180,E1 -1499.845,E2 -1499.845} C_VEL
LIN {X 0,Y 587.529,Z 487.752,A -85,B 0,C 180,E1 -1502.964,E2 -1502.964} C_VEL
LIN {X 0,Y 587.431,Z 498.623,A -85,B 0,C 180,E1 -1505.998,E2 -1505.998} C_VEL
LIN {X 0,Y 587.406,Z 508.136,A -85,B 0,C 180,E1 -1508.598,E2 -1508.598} C_VEL
LIN {X 0,Y 587.324,Z 519.006,A -85,B 0,C 180,E1 -1511.513,E2 -1511.513} C_VEL
LIN {X 0,Y 587.261,Z 529.877,A -85,B 0,C 180,E1 -1514.38,E2 -1514.38} C_VEL
LIN {X 0,Y 587.249,Z 540.748,A -85,B 0,C 180,E1 -1517.209,E2 -1517.209} C_VEL
LIN {X 0,Y 587.2,Z 551.619,A -85,B 0,C 180,E1 -1520.006,E2 -1520.006} C_VEL
LIN {X 0,Y 587.2,Z 552.978,A -85,B 0,C 180,E1 -1520.354,E2 -1520.354} C_VEL
LIN {X 0,Y 587.5,Z 561.258,A -85,B 0,C 180,E1 -1520.555,E2 -1520.555} C_VEL
LIN {X 0,Y 587.446,Z 571.307,A -85,B 0,C 180,E1 -1520.879,E2 -1520.879} C_VEL
LIN {X 0,Y 587.409,Z 582.742,A -85,B 0,C 180,E1 -1521.399,E2 -1521.399} C_VEL
LIN {X 0,Y 587.337,Z 592.551,A -85,B 0,C 180,E1 -1522.004,E2 -1522.004} C_VEL
LIN {X 0,Y 587.292,Z 600.406,A -85,B 0,C 180,E1 -1522.609,E2 -1522.609} C_VEL
LIN {X 0,Y 587.269,Z 608.288,A -85,B 0,C 180,E1 -1523.355,E2 -1523.355} C_VEL
LIN {X 0,Y 587.238,Z 616.434,A -85,B 0,C 180,E1 -1524.334,E2 -1524.334} C_VEL
LIN {X 0,Y 587.186,Z 621.988,A -85,B 0,C 180,E1 -1525.194,E2 -1525.194} C_VEL
LIN {X 0,Y 587.209,Z 627.149,A -85,B 0,C 180,E1 -1526.226,E2 -1526.226} C_VEL
LIN {X 0,Y 587.158,Z 629.789,A -85,B 0,C 180,E1 -1526.913,E2 -1526.913} C_VEL
LIN {X 0,Y 587.14,Z 632.681,A -85,B 0,C 180,E1 -1527.942,E2 -1527.942} C_VEL
LIN {X 0,Y 587.146,Z 633.936,A -85,B 0,C 180,E1 -1528.629,E2 -1528.629} C_VEL
LIN {X 0,Y 587.138,Z 634.712,A -85,B 0,C 180,E1 -1529.315,E2 -1529.315} C_VEL
LIN {X 0,Y 587.134,Z 635,A -85,B 0,C 180,E1 -1530,E2 -1530} C_VEL
LIN {X 0,Y 587.138,Z 634.712,A -85,B 0,C 180,E1 -1530.686,E2 -1530.686} C_VEL
LIN {X 0,Y 587.146,Z 633.935,A -85,B 0,C 180,E1 -1531.372,E2 -1531.372} C_VEL
LIN {X 0,Y 587.14,Z 632.679,A -85,B 0,C 180,E1 -1532.058,E2 -1532.058} C_VEL
LIN {X 0,Y 587.158,Z 629.786,A -85,B 0,C 180,E1 -1533.088,E2 -1533.088} C_VEL
LIN {X 0,Y 587.21,Z 627.145,A -85,B 0,C 180,E1 -1533.775,E2 -1533.775} C_VEL
LIN {X 0,Y 587.186,Z 621.983,A -85,B 0,C 180,E1 -1534.806,E2 -1534.806} C_VEL
LIN {X 0,Y 587.238,Z 616.428,A -85,B 0,C 180,E1 -1535.667,E2 -1535.667} C_VEL
LIN {X 0,Y 587.269,Z 608.284,A -85,B 0,C 180,E1 -1536.646,E2 -1536.646} C_VEL
LIN {X 0,Y 587.289,Z 601.414,A -85,B 0,C 180,E1 -1537.305,E2 -1537.305} C_VEL
LIN {X 0,Y 587.332,Z 593.761,A -85,B 0,C 180,E1 -1537.91,E2 -1537.91} C_VEL
LIN {X 0,Y 587.382,Z 585.72,A -85,B 0,C 180,E1 -1538.429,E2 -1538.429} C_VEL
LIN {X 0,Y 587.405,Z 577.389,A -85,B 0,C 180,E1 -1538.862,E2 -1538.862} C_VEL
LIN {X 0,Y 587.465,Z 568.882,A -85,B 0,C 180,E1 -1539.208,E2 -1539.208} C_VEL
LIN {X 0,Y 587.483,Z 558.741,A -85,B 0,C 180,E1 -1539.511,E2 -1539.511} C_VEL
LIN {X 0,Y 587.188,Z 553.301,A -85,B 0,C 180,E1 -1539.647,E2 -1539.647} C_VEL
LIN {X 0,Y 587.21,Z 543.082,A -85,B 0,C 180,E1 -1542.441,E2 -1542.441} C_VEL
LIN {X 0,Y 587.268,Z 532.864,A -85,B 0,C 180,E1 -1545.265,E2 -1545.265} C_VEL
LIN {X 0,Y 587.292,Z 522.645,A -85,B 0,C 180,E1 -1548.128,E2 -1548.128} C_VEL
LIN {X 0,Y 587.361,Z 512.397,A -85,B 0,C 180,E1 -1551.045,E2 -1551.045} C_VEL
LIN {X 0,Y 587.391,Z 502.207,A -85,B 0,C 180,E1 -1554.004,E2 -1554.004} C_VEL
LIN {X 0,Y 587.486,Z 493.266,A -85,B 0,C 180,E1 -1556.655,E2 -1556.655} C_VEL
LIN {X 0,Y 587.505,Z 484.243,A -85,B 0,C 180,E1 -1559.371,E2 -1559.371} C_VEL
LIN {X 0,Y 587.575,Z 476.24,A -85,B 0,C 180,E1 -1561.872,E2 -1561.872} C_VEL
LIN {X 0,Y 587.371,Z 472.152,A -85,B 0,C 180,E1 -1563.245,E2 -1563.245} C_VEL
LIN {X 0,Y 587.297,Z 472.142,A -85,B 0,C 180,E1 -1565.9,E2 -1565.9} C_VEL
LIN {X 0,Y 587.334,Z 472.14,A -85,B 0,C 180,E1 -1568.479,E2 -1568.479} C_VEL
LIN {X 0,Y 587.337,Z 472.135,A -85,B 0,C 180,E1 -1571.157,E2 -1571.157} C_VEL
LIN {X 0,Y 587.329,Z 472.136,A -85,B 0,C 180,E1 -1574.114,E2 -1574.114} C_VEL
LIN {X 0,Y 587.324,Z 472.138,A -85,B 0,C 180,E1 -1576.995,E2 -1576.995} C_VEL
LIN {X 0,Y 587.315,Z 472.143,A -85,B 0,C 180,E1 -1579.746,E2 -1579.746} C_VEL
LIN {X 0,Y 587.348,Z 472.134,A -85,B 0,C 180,E1 -1582.393,E2 -1582.393} C_VEL
LIN {X 0,Y 587.361,Z 472.134,A -85,B 0,C 180,E1 -1585.78,E2 -1585.78} C_VEL
LIN {X 0,Y 587.269,Z 472.334,A -85,B 0,C 180,E1 -1588.177,E2 -1588.177} C_VEL
LIN {X 0,Y 587.243,Z 476.191,A -85,B 0,C 180,E1 -1590.886,E2 -1590.886} C_VEL
LIN {X 0,Y 587.217,Z 480.302,A -85,B 0,C 180,E1 -1593.848,E2 -1593.848} C_VEL
LIN {X 0,Y 587.168,Z 484.698,A -85,B 0,C 180,E1 -1596.735,E2 -1596.735} C_VEL
LIN {X 0,Y 587.177,Z 489.293,A -85,B 0,C 180,E1 -1599.69,E2 -1599.69} C_VEL
LIN {X 0,Y 587.146,Z 492.739,A -85,B 0,C 180,E1 -1601.868,E2 -1601.868} C_VEL
LIN {X 0,Y 587.168,Z 497.334,A -85,B 0,C 180,E1 -1604.733,E2 -1604.733} C_VEL
LIN {X 0,Y 587.159,Z 501.93,A -85,B 0,C 180,E1 -1607.558,E2 -1607.558} C_VEL
LIN {X 0,Y 587.155,Z 506.705,A -85,B 0,C 180,E1 -1610.462,E2 -1610.462} C_VEL
LIN {X 0,Y 587.505,Z 512.847,A -85,B 0,C 180,E1 -1610.641,E2 -1610.641} C_VEL
LIN {X 0,Y 587.442,Z 524.563,A -85,B 0,C 180,E1 -1611.053,E2 -1611.053} C_VEL
LIN {X 0,Y 587.389,Z 534.955,A -85,B 0,C 180,E1 -1611.572,E2 -1611.572} C_VEL
LIN {X 0,Y 587.327,Z 543.133,A -85,B 0,C 180,E1 -1612.09,E2 -1612.09} C_VEL
LIN {X 0,Y 587.296,Z 550.891,A -85,B 0,C 180,E1 -1612.695,E2 -1612.695} C_VEL
LIN {X 0,Y 587.287,Z 558.731,A -85,B 0,C 180,E1 -1613.445,E2 -1613.445} C_VEL
LIN {X 0,Y 587.238,Z 566.123,A -85,B 0,C 180,E1 -1614.334,E2 -1614.334} C_VEL
LIN {X 0,Y 587.184,Z 571.735,A -85,B 0,C 180,E1 -1615.194,E2 -1615.194} C_VEL
LIN {X 0,Y 587.21,Z 576.949,A -85,B 0,C 180,E1 -1616.226,E2 -1616.226} C_VEL
LIN {X 0,Y 587.158,Z 579.637,A -85,B 0,C 180,E1 -1616.912,E2 -1616.912} C_VEL
LIN {X 0,Y 587.137,Z 582.575,A -85,B 0,C 180,E1 -1617.942,E2 -1617.942} C_VEL
LIN {X 0,Y 587.147,Z 583.874,A -85,B 0,C 180,E1 -1618.628,E2 -1618.628} C_VEL
LIN {X 0,Y 587.136,Z 584.691,A -85,B 0,C 180,E1 -1619.314,E2 -1619.314} C_VEL
LIN {X 0,Y 587.133,Z 584.996,A -85,B 0,C 180,E1 -1620,E2 -1620} C_VEL
LIN {X 0,Y 587.139,Z 584.733,A -85,B 0,C 180,E1 -1620.686,E2 -1620.686} C_VEL
LIN {X 0,Y 587.146,Z 583.997,A -85,B 0,C 180,E1 -1621.372,E2 -1621.372} C_VEL
LIN {X 0,Y 587.14,Z 582.785,A -85,B 0,C 180,E1 -1622.058,E2 -1622.058} C_VEL
LIN {X 0,Y 587.141,Z 579.938,A -85,B 0,C 180,E1 -1623.088,E2 -1623.088} C_VEL
LIN {X 0,Y 587.212,Z 577.345,A -85,B 0,C 180,E1 -1623.774,E2 -1623.774} C_VEL
LIN {X 0,Y 587.17,Z 572.236,A -85,B 0,C 180,E1 -1624.806,E2 -1624.806} C_VEL
LIN {X 0,Y 587.239,Z 566.739,A -85,B 0,C 180,E1 -1625.666,E2 -1625.666} C_VEL
LIN {X 0,Y 587.264,Z 558.799,A -85,B 0,C 180,E1 -1626.638,E2 -1626.638} C_VEL
LIN {X 0,Y 587.301,Z 550.929,A -85,B 0,C 180,E1 -1627.391,E2 -1627.391} C_VEL
LIN {X 0,Y 587.331,Z 543.179,A -85,B 0,C 180,E1 -1627.996,E2 -1627.996} C_VEL
LIN {X 0,Y 587.406,Z 535.01,A -85,B 0,C 180,E1 -1628.515,E2 -1628.515} C_VEL
LIN {X 0,Y 587.455,Z 524.63,A -85,B 0,C 180,E1 -1629.034,E2 -1629.034} C_VEL
LIN {X 0,Y 587.485,Z 512.962,A -85,B 0,C 180,E1 -1629.446,E2 -1629.446} C_VEL
LIN {X 0,Y 587.2,Z 507.146,A -85,B 0,C 180,E1 -1629.603,E2 -1629.603} C_VEL
LIN {X 0,Y 587.143,Z 506.484,A -85,B 0,C 180,E1 -1629.647,E2 -1629.647} C_VEL
LIN {X 0,Y 587.161,Z 501.593,A -85,B 0,C 180,E1 -1632.442,E2 -1632.442} C_VEL
LIN {X 0,Y 587.165,Z 497.436,A -85,B 0,C 180,E1 -1634.842,E2 -1634.842} C_VEL
LIN {X 0,Y 586.484,Z 496.494,A -85,B 0,C 180,E1 -1635.407,E2 -1635.407} C_VEL
LIN {X 0,Y 583.594,Z 495.062,A -85,B 0,C 180,E1 -1636.325,E2 -1636.325} C_VEL
LIN {X 0,Y 581.165,Z 493.931,A -85,B 0,C 180,E1 -1637.065,E2 -1637.065} C_VEL
LIN {X 0,Y 580.133,Z 493.024,A -85,B 0,C 180,E1 -1637.635,E2 -1637.635} C_VEL
LIN {X 0,Y 580.054,Z 492.705,A -85,B 0,C 180,E1 -1637.828,E2 -1637.828} C_VEL
LIN {X 0,Y 580.093,Z 488.142,A -85,B 0,C 180,E1 -1640.57,E2 -1640.57} C_VEL
LIN {X 0,Y 580.12,Z 483.251,A -85,B 0,C 180,E1 -1643.565,E2 -1643.565} C_VEL
LIN {X 0,Y 580.145,Z 478.397,A -85,B 0,C 180,E1 -1646.63,E2 -1646.63} C_VEL
LIN {X 0,Y 580.197,Z 477.497,A -85,B 0,C 180,E1 -1647.309,E2 -1647.309} C_VEL
LIN {X 0,Y 580.206,Z 483.819,A -85,B 0,C 180,E1 -1649.777,E2 -1649.777} C_VEL
LIN {X 0,Y 580.233,Z 489.648,A -85,B 0,C 180,E1 -1652.205,E2 -1652.205} C_VEL
LIN {X 0,Y 580.183,Z 496.74,A -85,B 0,C 180,E1 -1655.127,E2 -1655.127} C_VEL
LIN {X 0,Y 580.137,Z 504.242,A -85,B 0,C 180,E1 -1658.158,E2 -1658.158} C_VEL
LIN {X 0,Y 580.115,Z 511.035,A -85,B 0,C 180,E1 -1660.859,E2 -1660.859} C_VEL
LIN {X 0,Y 580.105,Z 518.206,A -85,B 0,C 180,E1 -1663.674,E2 -1663.674} C_VEL
LIN {X 0,Y 580.088,Z 525.026,A -85,B 0,C 180,E1 -1666.324,E2 -1666.324} C_VEL
LIN {X 0,Y 580.497,Z 531.771,A -85,B 0,C 180,E1 -1666.498,E2 -1666.498} C_VEL
LIN {X 0,Y 580.458,Z 541.891,A -85,B 0,C 180,E1 -1666.836,E2 -1666.836} C_VEL
LIN {X 0,Y 580.365,Z 553.768,A -85,B 0,C 180,E1 -1667.397,E2 -1667.397} C_VEL
LIN {X 0,Y 580.304,Z 563.326,A -85,B 0,C 180,E1 -1668.005,E2 -1668.005} C_VEL
LIN {X 0,Y 580.254,Z 571.695,A -85,B 0,C 180,E1 -1668.672,E2 -1668.672} C_VEL
LIN {X 0,Y 580.157,Z 579.701,A -85,B 0,C 180,E1 -1669.47,E2 -1669.47} C_VEL
LIN {X 0,Y 580.159,Z 586.115,A -85,B 0,C 180,E1 -1670.265,E2 -1670.265} C_VEL
LIN {X 0,Y 580.143,Z 591.993,A -85,B 0,C 180,E1 -1671.177,E2 -1671.177} C_VEL
LIN {X 0,Y 580.097,Z 595.98,A -85,B 0,C 180,E1 -1671.952,E2 -1671.952} C_VEL
LIN {X 0,Y 580.059,Z 600.392,A -85,B 0,C 180,E1 -1673.097,E2 -1673.097} C_VEL
LIN {X 0,Y 580.029,Z 603.376,A -85,B 0,C 180,E1 -1674.274,E2 -1674.274} C_VEL
LIN {X 0,Y 580.048,Z 604.769,A -85,B 0,C 180,E1 -1675.478,E2 -1675.478} C_VEL
LIN {X 0,Y 580.044,Z 604.986,A -85,B 0,C 180,E1 -1676.127,E2 -1676.127} C_VEL
LIN {X 0,Y 580.045,Z 604.569,A -85,B 0,C 180,E1 -1676.959,E2 -1676.959} C_VEL
LIN {X 0,Y 580.043,Z 602.964,A -85,B 0,C 180,E1 -1678.01,E2 -1678.01} C_VEL
LIN {X 0,Y 580.081,Z 600.372,A -85,B 0,C 180,E1 -1678.999,E2 -1678.999} C_VEL
LIN {X 0,Y 580.086,Z 597.392,A -85,B 0,C 180,E1 -1679.815,E2 -1679.815} C_VEL
LIN {X 0,Y 580.1,Z 593.024,A -85,B 0,C 180,E1 -1680.726,E2 -1680.726} C_VEL
LIN {X 0,Y 580.133,Z 587.628,A -85,B 0,C 180,E1 -1681.608,E2 -1681.608} C_VEL
LIN {X 0,Y 580.206,Z 581.777,A -85,B 0,C 180,E1 -1682.379,E2 -1682.379} C_VEL
LIN {X 0,Y 580.213,Z 573.26,A -85,B 0,C 180,E1 -1683.276,E2 -1683.276} C_VEL
LIN {X 0,Y 580.305,Z 564.478,A -85,B 0,C 180,E1 -1684.002,E2 -1684.002} C_VEL
LIN {X 0,Y 580.382,Z 554.739,A -85,B 0,C 180,E1 -1684.636,E2 -1684.636} C_VEL
LIN {X 0,Y 580.448,Z 543.81,A -85,B 0,C 180,E1 -1685.18,E2 -1685.18} C_VEL
LIN {X 0,Y 580.505,Z 532.404,A -85,B 0,C 180,E1 -1685.575,E2 -1685.575} C_VEL
LIN {X 0,Y 580.116,Z 526.044,A -85,B 0,C 180,E1 -1685.747,E2 -1685.747} C_VEL
LIN {X 0,Y 580.056,Z 525.277,A -85,B 0,C 180,E1 -1685.768,E2 -1685.768} C_VEL
LIN {X 0,Y 580.045,Z 520.023,A -85,B 0,C 180,E1 -1687.938,E2 -1687.938} C_VEL
LIN {X 0,Y 580.137,Z 512.896,A -85,B 0,C 180,E1 -1690.908,E2 -1690.908} C_VEL
LIN {X 0,Y 580.146,Z 506.001,A -85,B 0,C 180,E1 -1693.821,E2 -1693.821} C_VEL
LIN {X 0,Y 580.144,Z 499.317,A -85,B 0,C 180,E1 -1696.693,E2 -1696.693} C_VEL
LIN {X 0,Y 580.198,Z 492.827,A -85,B 0,C 180,E1 -1699.531,E2 -1699.531} C_VEL
LIN {X 0,Y 580.217,Z 486.481,A -85,B 0,C 180,E1 -1702.343,E2 -1702.343} C_VEL
LIN {X 0,Y 580.242,Z 479.914,A -85,B 0,C 180,E1 -1705.136,E2 -1705.136} C_VEL
LIN {X 0,Y 580.259,Z 473.022,A -85,B 0,C 180,E1 -1708.091,E2 -1708.091} C_VEL
LIN {X 0,Y 580.357,Z 473.007,A -85,B 0,C 180,E1 -1710,E2 -1710} C_VEL
LIN {X 0,Y 580.339,Z 473.011,A -85,B 0,C 180,E1 -1712.776,E2 -1712.776} C_VEL
LIN {X 0,Y 580.333,Z 473.011,A -85,B 0,C 180,E1 -1715.559,E2 -1715.559} C_VEL
LIN {X 0,Y 580.331,Z 473.01,A -85,B 0,C 180,E1 -1718.356,E2 -1718.356} C_VEL
LIN {X 0,Y 580.302,Z 473.017,A -85,B 0,C 180,E1 -1721.191,E2 -1721.191} C_VEL
LIN {X 0,Y 580.328,Z 473.011,A -85,B 0,C 180,E1 -1724.017,E2 -1724.017} C_VEL
LIN {X 0,Y 580.313,Z 473.014,A -85,B 0,C 180,E1 -1726.913,E2 -1726.913} C_VEL
LIN {X 0,Y 580.307,Z 473.014,A -85,B 0,C 180,E1 -1729.822,E2 -1729.822} C_VEL
LIN {X 0,Y 580.296,Z 473.016,A -85,B 0,C 180,E1 -1732.802,E2 -1732.802} C_VEL
LIN {X 0,Y 580.31,Z 473.014,A -85,B 0,C 180,E1 -1735.079,E2 -1735.079} C_VEL
LIN {X 0,Y 580.299,Z 473.016,A -85,B 0,C 180,E1 -1737.859,E2 -1737.859} C_VEL
LIN {X 0,Y 580.301,Z 473.014,A -85,B 0,C 180,E1 -1740.697,E2 -1740.697} C_VEL
LIN {X 0,Y 580.305,Z 473.014,A -85,B 0,C 180,E1 -1743.316,E2 -1743.316} C_VEL
LIN {X 0,Y 580.326,Z 473.012,A -85,B 0,C 180,E1 -1745.767,E2 -1745.767} C_VEL
LIN {X 0,Y 580.29,Z 473.017,A -85,B 0,C 180,E1 -1748.146,E2 -1748.146} C_VEL
LIN {X 0,Y 580.298,Z 473.016,A -85,B 0,C 180,E1 -1750.843,E2 -1750.843} C_VEL
LIN {X 0,Y 580.287,Z 473.015,A -85,B 0,C 180,E1 -1753.657,E2 -1753.657} C_VEL
LIN {X 0,Y 580.285,Z 473.019,A -85,B 0,C 180,E1 -1756.608,E2 -1756.608} C_VEL
LIN {X 0,Y 580.32,Z 473.013,A -85,B 0,C 180,E1 -1759.158,E2 -1759.158} C_VEL
LIN {X 0,Y 580.29,Z 473.015,A -85,B 0,C 180,E1 -1761.926,E2 -1761.926} C_VEL
LIN {X 0,Y 580.251,Z 473.02,A -85,B 0,C 180,E1 -1764.453,E2 -1764.453} C_VEL
LIN {X 0,Y 580.292,Z 473.016,A -85,B 0,C 180,E1 -1766.975,E2 -1766.975} C_VEL
LIN {X 0,Y 580.3,Z 473.015,A -85,B 0,C 180,E1 -1769.425,E2 -1769.425} C_VEL
LIN {X 0,Y 580.319,Z 473.013,A -85,B 0,C 180,E1 -1772.137,E2 -1772.137} C_VEL
LIN {X 0,Y 580.308,Z 473.012,A -85,B 0,C 180,E1 -1774.92,E2 -1774.92} C_VEL
LIN {X 0,Y 580.275,Z 473.02,A -85,B 0,C 180,E1 -1777.947,E2 -1777.947} C_VEL
LIN {X 0,Y 580.317,Z 473.011,A -85,B 0,C 180,E1 -1780.914,E2 -1780.914} C_VEL
LIN {X 0,Y 580.282,Z 473.019,A -85,B 0,C 180,E1 -1783.826,E2 -1783.826} C_VEL
LIN {X 0,Y 580.326,Z 473.013,A -85,B 0,C 180,E1 -1785.983,E2 -1785.983} C_VEL
LIN {X 0,Y 580.302,Z 473.014,A -85,B 0,C 180,E1 -1788.827,E2 -1788.827} C_VEL
LIN {X 0,Y 580.334,Z 473.01,A -85,B 0,C 180,E1 -1791.644,E2 -1791.644} C_VEL
LIN {X 0,Y 580.322,Z 473.014,A -85,B 0,C 180,E1 -1794.44,E2 -1794.44} C_VEL
LIN {X 0,Y 580.345,Z 473.008,A -85,B 0,C 180,E1 -1797.223,E2 -1797.223} C_VEL
LIN {X 0,Y 580.351,Z 473.008,A -85,B 0,C 180,E1 -1800,E2 -1800} C_VEL
LIN {X 0,Y 580.344,Z 473.011,A -85,B 0,C 180,E1 -1802.776,E2 -1802.776} C_VEL
LIN {X 0,Y 580.328,Z 473.011,A -85,B 0,C 180,E1 -1805.56,E2 -1805.56} C_VEL
LIN {X 0,Y 580.332,Z 473.011,A -85,B 0,C 180,E1 -1808.356,E2 -1808.356} C_VEL
LIN {X 0,Y 580.298,Z 473.016,A -85,B 0,C 180,E1 -1811.191,E2 -1811.191} C_VEL
LIN {X 0,Y 580.324,Z 473.011,A -85,B 0,C 180,E1 -1814.017,E2 -1814.017} C_VEL
LIN {X 0,Y 580.312,Z 473.016,A -85,B 0,C 180,E1 -1816.915,E2 -1816.915} C_VEL
LIN {X 0,Y 580.304,Z 473.013,A -85,B 0,C 180,E1 -1819.822,E2 -1819.822} C_VEL
LIN {X 0,Y 580.296,Z 473.017,A -85,B 0,C 180,E1 -1822.802,E2 -1822.802} C_VEL
LIN {X 0,Y 580.305,Z 473.016,A -85,B 0,C 180,E1 -1825.08,E2 -1825.08} C_VEL
LIN {X 0,Y 580.299,Z 473.014,A -85,B 0,C 180,E1 -1828.185,E2 -1828.185} C_VEL
LIN {X 0,Y 580.297,Z 473.014,A -85,B 0,C 180,E1 -1830.697,E2 -1830.697} C_VEL
LIN {X 0,Y 580.303,Z 473.016,A -85,B 0,C 180,E1 -1833.317,E2 -1833.317} C_VEL
LIN {X 0,Y 580.325,Z 473.014,A -85,B 0,C 180,E1 -1835.768,E2 -1835.768} C_VEL
LIN {X 0,Y 580.287,Z 473.018,A -85,B 0,C 180,E1 -1838.146,E2 -1838.146} C_VEL
LIN {X 0,Y 580.298,Z 473.015,A -85,B 0,C 180,E1 -1840.843,E2 -1840.843} C_VEL
LIN {X 0,Y 580.29,Z 473.016,A -85,B 0,C 180,E1 -1843.657,E2 -1843.657} C_VEL
LIN {X 0,Y 580.276,Z 473.018,A -85,B 0,C 180,E1 -1846.609,E2 -1846.609} C_VEL
LIN {X 0,Y 580.305,Z 473.014,A -85,B 0,C 180,E1 -1849.158,E2 -1849.158} C_VEL
LIN {X 0,Y 580.289,Z 473.016,A -85,B 0,C 180,E1 -1851.927,E2 -1851.927} C_VEL
LIN {X 0,Y 580.307,Z 473.015,A -85,B 0,C 180,E1 -1854.457,E2 -1854.457} C_VEL
LIN {X 0,Y 580.29,Z 473.019,A -85,B 0,C 180,E1 -1856.976,E2 -1856.976} C_VEL
LIN {X 0,Y 580.347,Z 473.152,A -85,B 0,C 180,E1 -1858.314,E2 -1858.314} C_VEL
LIN {X 0,Y 580.626,Z 476.839,A -85,B 0,C 180,E1 -1859.445,E2 -1859.445} C_VEL
LIN {X 0,Y 580.527,Z 485.916,A -85,B 0,C 180,E1 -1862.099,E2 -1862.099} C_VEL
LIN {X 0,Y 580.453,Z 495.905,A -85,B 0,C 180,E1 -1864.927,E2 -1864.927} C_VEL
LIN {X 0,Y 580.393,Z 506.776,A -85,B 0,C 180,E1 -1867.953,E2 -1867.953} C_VEL
LIN {X 0,Y 580.3,Z 517.647,A -85,B 0,C 180,E1 -1870.914,E2 -1870.914} C_VEL
LIN {X 0,Y 580.234,Z 528.518,A -85,B 0,C 180,E1 -1873.825,E2 -1873.825} C_VEL
LIN {X 0,Y 580.175,Z 539.389,A -85,B 0,C 180,E1 -1876.694,E2 -1876.694} C_VEL
LIN {X 0,Y 580.156,Z 549.007,A -85,B 0,C 180,E1 -1879.205,E2 -1879.205} C_VEL
LIN {X 0,Y 580.14,Z 552.978,A -85,B 0,C 180,E1 -1880.236,E2 -1880.236} C_VEL
LIN {X 0,Y 580.513,Z 560.428,A -85,B 0,C 180,E1 -1880.418,E2 -1880.418} C_VEL
LIN {X 0,Y 580.464,Z 568.902,A -85,B 0,C 180,E1 -1880.681,E2 -1880.681} C_VEL
LIN {X 0,Y 580.409,Z 577.406,A -85,B 0,C 180,E1 -1881.031,E2 -1881.031} C_VEL
LIN {X 0,Y 580.363,Z 585.734,A -85,B 0,C 180,E1 -1881.469,E2 -1881.469} C_VEL
LIN {X 0,Y 580.307,Z 593.771,A -85,B 0,C 180,E1 -1881.995,E2 -1881.995} C_VEL
LIN {X 0,Y 580.237,Z 601.42,A -85,B 0,C 180,E1 -1882.606,E2 -1882.606} C_VEL
LIN {X 0,Y 580.206,Z 609.766,A -85,B 0,C 180,E1 -1883.428,E2 -1883.428} C_VEL
LIN {X 0,Y 580.173,Z 616.435,A -85,B 0,C 180,E1 -1884.265,E2 -1884.265} C_VEL
LIN {X 0,Y 580.097,Z 621.989,A -85,B 0,C 180,E1 -1885.135,E2 -1885.135} C_VEL
LIN {X 0,Y 580.136,Z 627.149,A -85,B 0,C 180,E1 -1886.18,E2 -1886.18} C_VEL
LIN {X 0,Y 580.073,Z 629.789,A -85,B 0,C 180,E1 -1886.875,E2 -1886.875} C_VEL
LIN {X 0,Y 580.039,Z 632.681,A -85,B 0,C 180,E1 -1887.917,E2 -1887.917} C_VEL
LIN {X 0,Y 580.045,Z 633.936,A -85,B 0,C 180,E1 -1888.612,E2 -1888.612} C_VEL
LIN {X 0,Y 580.038,Z 634.712,A -85,B 0,C 180,E1 -1889.306,E2 -1889.306} C_VEL
LIN {X 0,Y 580.034,Z 635,A -85,B 0,C 180,E1 -1890,E2 -1890} C_VEL
LIN {X 0,Y 580.038,Z 634.711,A -85,B 0,C 180,E1 -1890.695,E2 -1890.695} C_VEL
LIN {X 0,Y 580.045,Z 633.935,A -85,B 0,C 180,E1 -1891.389,E2 -1891.389} C_VEL
LIN {X 0,Y 580.039,Z 632.679,A -85,B 0,C 180,E1 -1892.083,E2 -1892.083} C_VEL
LIN {X 0,Y 580.073,Z 629.786,A -85,B 0,C 180,E1 -1893.126,E2 -1893.126} C_VEL
LIN {X 0,Y 580.122,Z 627.146,A -85,B 0,C 180,E1 -1893.821,E2 -1893.821} C_VEL
LIN {X 0,Y 580.097,Z 621.983,A -85,B 0,C 180,E1 -1894.865,E2 -1894.865} C_VEL
LIN {X 0,Y 580.173,Z 616.428,A -85,B 0,C 180,E1 -1895.736,E2 -1895.736} C_VEL
LIN {X 0,Y 580.209,Z 608.946,A -85,B 0,C 180,E1 -1896.659,E2 -1896.659} C_VEL
LIN {X 0,Y 580.238,Z 601.415,A -85,B 0,C 180,E1 -1897.394,E2 -1897.394} C_VEL
LIN {X 0,Y 580.308,Z 593.763,A -85,B 0,C 180,E1 -1898.006,E2 -1898.006} C_VEL
LIN {X 0,Y 580.363,Z 585.722,A -85,B 0,C 180,E1 -1898.531,E2 -1898.531} C_VEL
LIN {X 0,Y 580.408,Z 577.391,A -85,B 0,C 180,E1 -1898.969,E2 -1898.969} C_VEL
LIN {X 0,Y 580.47,Z 568.884,A -85,B 0,C 180,E1 -1899.32,E2 -1899.32} C_VEL
LIN {X 0,Y 580.496,Z 558.74,A -85,B 0,C 180,E1 -1899.627,E2 -1899.627} C_VEL
LIN {X 0,Y 580.096,Z 553.301,A -85,B 0,C 180,E1 -1899.766,E2 -1899.766} C_VEL
LIN {X 0,Y 580.152,Z 543.082,A -85,B 0,C 180,E1 -1902.595,E2 -1902.595} C_VEL
LIN {X 0,Y 580.217,Z 534.141,A -85,B 0,C 180,E1 -1905.096,E2 -1905.096} C_VEL
LIN {X 0,Y 580.253,Z 523.922,A -85,B 0,C 180,E1 -1907.991,E2 -1907.991} C_VEL
LIN {X 0,Y 580.304,Z 513.933,A -85,B 0,C 180,E1 -1910.866,E2 -1910.866} C_VEL
LIN {X 0,Y 580.372,Z 504.762,A -85,B 0,C 180,E1 -1913.554,E2 -1913.554} C_VEL
LIN {X 0,Y 580.456,Z 495.361,A -85,B 0,C 180,E1 -1916.367,E2 -1916.367} C_VEL
LIN {X 0,Y 580.494,Z 486.755,A -85,B 0,C 180,E1 -1918.965,E2 -1918.965} C_VEL
LIN {X 0,Y 580.604,Z 479.076,A -85,B 0,C 180,E1 -1921.366,E2 -1921.366} C_VEL
LIN {X 0,Y 580.502,Z 474.183,A -85,B 0,C 180,E1 -1923.012,E2 -1923.012} C_VEL
LIN {X 0,Y 580.323,Z 473.014,A -85,B 0,C 180,E1 -1923.442,E2 -1923.442} C_VEL
LIN {X 0,Y 580.272,Z 473.016,A -85,B 0,C 180,E1 -1926.404,E2 -1926.404} C_VEL
LIN {X 0,Y 580.31,Z 473.011,A -85,B 0,C 180,E1 -1929.187,E2 -1929.187} C_VEL
LIN {X 0,Y 580.282,Z 473.019,A -85,B 0,C 180,E1 -1931.769,E2 -1931.769} C_VEL
LIN {X 0,Y 580.27,Z 473.017,A -85,B 0,C 180,E1 -1934.626,E2 -1934.626} C_VEL
LIN {X 0,Y 580.284,Z 473.013,A -85,B 0,C 180,E1 -1937.294,E2 -1937.294} C_VEL
LIN {X 0,Y 580.287,Z 473.016,A -85,B 0,C 180,E1 -1940.067,E2 -1940.067} C_VEL
LIN {X 0,Y 580.302,Z 473.017,A -85,B 0,C 180,E1 -1943.066,E2 -1943.066} C_VEL
LIN {X 0,Y 580.318,Z 473.015,A -85,B 0,C 180,E1 -1946.145,E2 -1946.145} C_VEL
LIN {X 0,Y 580.229,Z 473.026,A -85,B 0,C 180,E1 -1947.982,E2 -1947.982} C_VEL
LIN {X 0,Y 580.161,Z 475.972,A -85,B 0,C 180,E1 -1950.22,E2 -1950.22} C_VEL
LIN {X 0,Y 580.127,Z 479.193,A -85,B 0,C 180,E1 -1952.59,E2 -1952.59} C_VEL
LIN {X 0,Y 580.092,Z 482.401,A -85,B 0,C 180,E1 -1954.91,E2 -1954.91} C_VEL
LIN {X 0,Y 580.098,Z 485.848,A -85,B 0,C 180,E1 -1957.189,E2 -1957.189} C_VEL
LIN {X 0,Y 580.092,Z 489.294,A -85,B 0,C 180,E1 -1959.431,E2 -1959.431} C_VEL
LIN {X 0,Y 580.09,Z 492.74,A -85,B 0,C 180,E1 -1961.639,E2 -1961.639} C_VEL
LIN {X 0,Y 580.077,Z 497.335,A -85,B 0,C 180,E1 -1964.541,E2 -1964.541} C_VEL
LIN {X 0,Y 580.061,Z 500.782,A -85,B 0,C 180,E1 -1966.691,E2 -1966.691} C_VEL
LIN {X 0,Y 580.054,Z 505.377,A -85,B 0,C 180,E1 -1969.529,E2 -1969.529} C_VEL
LIN {X 0,Y 580.06,Z 506.706,A -85,B 0,C 180,E1 -1970.344,E2 -1970.344} C_VEL
LIN {X 0,Y 580.504,Z 512.038,A -85,B 0,C 180,E1 -1970.505,E2 -1970.505} C_VEL
LIN {X 0,Y 580.444,Z 523.59,A -85,B 0,C 180,E1 -1970.9,E2 -1970.9} C_VEL
LIN {X 0,Y 580.354,Z 533.466,A -85,B 0,C 180,E1 -1971.381,E2 -1971.381} C_VEL
LIN {X 0,Y 580.29,Z 541.918,A -85,B 0,C 180,E1 -1971.906,E2 -1971.906} C_VEL
LIN {X 0,Y 580.26,Z 549.885,A -85,B 0,C 180,E1 -1972.519,E2 -1972.519} C_VEL
LIN {X 0,Y 580.23,Z 557.034,A -85,B 0,C 180,E1 -1973.19,E2 -1973.19} C_VEL
LIN {X 0,Y 580.209,Z 563.414,A -85,B 0,C 180,E1 -1973.916,E2 -1973.916} C_VEL
LIN {X 0,Y 580.091,Z 569.654,A -85,B 0,C 180,E1 -1974.787,E2 -1974.787} C_VEL
LIN {X 0,Y 580.105,Z 575.435,A -85,B 0,C 180,E1 -1975.832,E2 -1975.832} C_VEL
LIN {X 0,Y 580.123,Z 578.449,A -85,B 0,C 180,E1 -1976.527,E2 -1976.527} C_VEL
LIN {X 0,Y 580.047,Z 580.785,A -85,B 0,C 180,E1 -1977.222,E2 -1977.222} C_VEL
LIN {X 0,Y 580.037,Z 582.577,A -85,B 0,C 180,E1 -1977.917,E2 -1977.917} C_VEL
LIN {X 0,Y 580.047,Z 583.875,A -85,B 0,C 180,E1 -1978.611,E2 -1978.611} C_VEL
LIN {X 0,Y 580.037,Z 584.691,A -85,B 0,C 180,E1 -1979.306,E2 -1979.306} C_VEL
LIN {X 0,Y 580.034,Z 584.996,A -85,B 0,C 180,E1 -1980,E2 -1980} C_VEL
LIN {X 0,Y 580.039,Z 584.732,A -85,B 0,C 180,E1 -1980.694,E2 -1980.694} C_VEL
LIN {X 0,Y 580.045,Z 583.997,A -85,B 0,C 180,E1 -1981.389,E2 -1981.389} C_VEL
LIN {X 0,Y 580.039,Z 582.784,A -85,B 0,C 180,E1 -1982.083,E2 -1982.083} C_VEL
LIN {X 0,Y 580.059,Z 579.936,A -85,B 0,C 180,E1 -1983.125,E2 -1983.125} C_VEL
LIN {X 0,Y 580.124,Z 577.343,A -85,B 0,C 180,E1 -1983.821,E2 -1983.821} C_VEL
LIN {X 0,Y 580.076,Z 572.234,A -85,B 0,C 180,E1 -1984.865,E2 -1984.865} C_VEL
LIN {X 0,Y 580.173,Z 566.736,A -85,B 0,C 180,E1 -1985.736,E2 -1985.736} C_VEL
LIN {X 0,Y 580.196,Z 559.51,A -85,B 0,C 180,E1 -1986.645,E2 -1986.645} C_VEL
LIN {X 0,Y 580.257,Z 550.923,A -85,B 0,C 180,E1 -1987.481,E2 -1987.481} C_VEL
LIN {X 0,Y 580.297,Z 543.173,A -85,B 0,C 180,E1 -1988.094,E2 -1988.094} C_VEL
LIN {X 0,Y 580.395,Z 535.003,A -85,B 0,C 180,E1 -1988.618,E2 -1988.618} C_VEL
LIN {X 0,Y 580.434,Z 524.616,A -85,B 0,C 180,E1 -1989.144,E2 -1989.144} C_VEL
LIN {X 0,Y 580.483,Z 512.941,A -85,B 0,C 180,E1 -1989.561,E2 -1989.561} C_VEL
LIN {X 0,Y 580.108,Z 507.124,A -85,B 0,C 180,E1 -1989.721,E2 -1989.721} C_VEL
LIN {X 0,Y 580.05,Z 506.483,A -85,B 0,C 180,E1 -1989.766,E2 -1989.766} C_VEL
LIN {X 0,Y 580.072,Z 501.592,A -85,B 0,C 180,E1 -1992.597,E2 -1992.597} C_VEL
LIN {X 0,Y 580.077,Z 497.748,A -85,B 0,C 180,E1 -1994.843,E2 -1994.843} C_VEL
LIN {X 0,Y 580.054,Z 493.033,A -85,B 0,C 180,E1 -1997.632,E2 -1997.632} C_VEL
LIN {X 0,Y 580.054,Z 492.705,A -85,B 0,C 180,E1 -1997.828,E2 -1997.828} C_VEL
LIN {X 0,Y 579.399,Z 491.783,A -85,B 0,C 180,E1 -1998.4,E2 -1998.4} C_VEL
LIN {X 0,Y 576.54,Z 490.398,A -85,B 0,C 180,E1 -1999.33,E2 -1999.33} C_VEL
LIN {X 0,Y 574.118,Z 489.308,A -85,B 0,C 180,E1 -2000.079,E2 -2000.079} C_VEL
LIN {X 0,Y 573.082,Z 488.428,A -85,B 0,C 180,E1 -2000.657,E2 -2000.657} C_VEL
LIN {X 0,Y 573,Z 488.115,A -85,B 0,C 180,E1 -2000.852,E2 -2000.852} C_VEL
LIN {X 0,Y 573.035,Z 483.25,A -85,B 0,C 180,E1 -2003.874,E2 -2003.874} C_VEL
LIN {X 0,Y 573.088,Z 478.509,A -85,B 0,C 180,E1 -2006.984,E2 -2006.984} C_VEL
LIN {X 0,Y 573.108,Z 478.083,A -85,B 0,C 180,E1 -2007.279,E2 -2007.279} C_VEL
LIN {X 0,Y 573.141,Z 483.525,A -85,B 0,C 180,E1 -2009.469,E2 -2009.469} C_VEL
LIN {X 0,Y 573.168,Z 490.41,A -85,B 0,C 180,E1 -2012.214,E2 -2012.214} C_VEL
LIN {X 0,Y 573.101,Z 496.487,A -85,B 0,C 180,E1 -2014.751,E2 -2014.751} C_VEL
LIN {X 0,Y 573.082,Z 502.307,A -85,B 0,C 180,E1 -2017.143,E2 -2017.143} C_VEL
LIN {X 0,Y 573.071,Z 509.517,A -85,B 0,C 180,E1 -2020.059,E2 -2020.059} C_VEL
LIN {X 0,Y 573.021,Z 515.929,A -85,B 0,C 180,E1 -2022.617,E2 -2022.617} C_VEL
LIN {X 0,Y 573.038,Z 522.836,A -85,B 0,C 180,E1 -2025.344,E2 -2025.344} C_VEL
LIN {X 0,Y 573.016,Z 524.991,A -85,B 0,C 180,E1 -2026.189,E2 -2026.189} C_VEL
LIN {X 0,Y 573.489,Z 531.619,A -85,B 0,C 180,E1 -2026.376,E2 -2026.376} C_VEL
LIN {X 0,Y 573.446,Z 541.499,A -85,B 0,C 180,E1 -2026.708,E2 -2026.708} C_VEL
LIN {X 0,Y 573.338,Z 552.551,A -85,B 0,C 180,E1 -2027.219,E2 -2027.219} C_VEL
LIN {X 0,Y 573.262,Z 562.153,A -85,B 0,C 180,E1 -2027.82,E2 -2027.82} C_VEL
LIN {X 0,Y 573.199,Z 571.235,A -85,B 0,C 180,E1 -2028.54,E2 -2028.54} C_VEL
LIN {X 0,Y 573.088,Z 579.314,A -85,B 0,C 180,E1 -2029.345,E2 -2029.345} C_VEL
LIN {X 0,Y 573.088,Z 585.858,A -85,B 0,C 180,E1 -2030.159,E2 -2030.159} C_VEL
LIN {X 0,Y 573.051,Z 590.951,A -85,B 0,C 180,E1 -2030.936,E2 -2030.936} C_VEL
LIN {X 0,Y 573.026,Z 596.192,A -85,B 0,C 180,E1 -2031.949,E2 -2031.949} C_VEL
LIN {X 0,Y 572.979,Z 600.383,A -85,B 0,C 180,E1 -2033.057,E2 -2033.057} C_VEL
LIN {X 0,Y 572.93,Z 602.973,A -85,B 0,C 180,E1 -2034.058,E2 -2034.058} C_VEL
LIN {X 0,Y 572.961,Z 604.669,A -85,B 0,C 180,E1 -2035.268,E2 -2035.268} C_VEL
LIN {X 0,Y 572.939,Z 604.812,A -85,B 0,C 180,E1 -2036.525,E2 -2036.525} C_VEL
LIN {X 0,Y 572.951,Z 603.405,A -85,B 0,C 180,E1 -2037.82,E2 -2037.82} C_VEL
LIN {X 0,Y 572.996,Z 600.515,A -85,B 0,C 180,E1 -2038.992,E2 -2038.992} C_VEL
LIN {X 0,Y 572.989,Z 597.626,A -85,B 0,C 180,E1 -2039.809,E2 -2039.809} C_VEL
LIN {X 0,Y 573.03,Z 592.823,A -85,B 0,C 180,E1 -2040.822,E2 -2040.822} C_VEL
LIN {X 0,Y 573.06,Z 587.19,A -85,B 0,C 180,E1 -2041.744,E2 -2041.744} C_VEL
LIN {X 0,Y 573.148,Z 580.372,A -85,B 0,C 180,E1 -2042.624,E2 -2042.624} C_VEL
LIN {X 0,Y 573.165,Z 572.463,A -85,B 0,C 180,E1 -2043.439,E2 -2043.439} C_VEL
LIN {X 0,Y 573.266,Z 564.449,A -85,B 0,C 180,E1 -2044.103,E2 -2044.103} C_VEL
LIN {X 0,Y 573.329,Z 556.037,A -85,B 0,C 180,E1 -2044.665,E2 -2044.665} C_VEL
LIN {X 0,Y 573.369,Z 546.213,A -85,B 0,C 180,E1 -2045.184,E2 -2045.184} C_VEL
LIN {X 0,Y 573.517,Z 534.196,A -85,B 0,C 180,E1 -2045.642,E2 -2045.642} C_VEL
LIN {X 0,Y 573.263,Z 527.712,A -85,B 0,C 180,E1 -2045.823,E2 -2045.823} C_VEL
LIN {X 0,Y 572.967,Z 525.236,A -85,B 0,C 180,E1 -2045.906,E2 -2045.906} C_VEL
LIN {X 0,Y 572.988,Z 518.38,A -85,B 0,C 180,E1 -2048.777,E2 -2048.777} C_VEL
LIN {X 0,Y 573.034,Z 512.171,A -85,B 0,C 180,E1 -2051.405,E2 -2051.405} C_VEL
LIN {X 0,Y 573.064,Z 505.311,A -85,B 0,C 180,E1 -2054.347,E2 -2054.347} C_VEL
LIN {X 0,Y 573.067,Z 500.307,A -85,B 0,C 180,E1 -2056.525,E2 -2056.525} C_VEL
LIN {X 0,Y 573.126,Z 493.805,A -85,B 0,C 180,E1 -2059.4,E2 -2059.4} C_VEL
LIN {X 0,Y 573.13,Z 488.912,A -85,B 0,C 180,E1 -2061.538,E2 -2061.538} C_VEL
LIN {X 0,Y 573.169,Z 483.935,A -85,B 0,C 180,E1 -2063.664,E2 -2063.664} C_VEL
LIN {X 0,Y 573.183,Z 479.049,A -85,B 0,C 180,E1 -2065.781,E2 -2065.781} C_VEL
